Yaskawa INFORM job: miniTRJ1.JBI

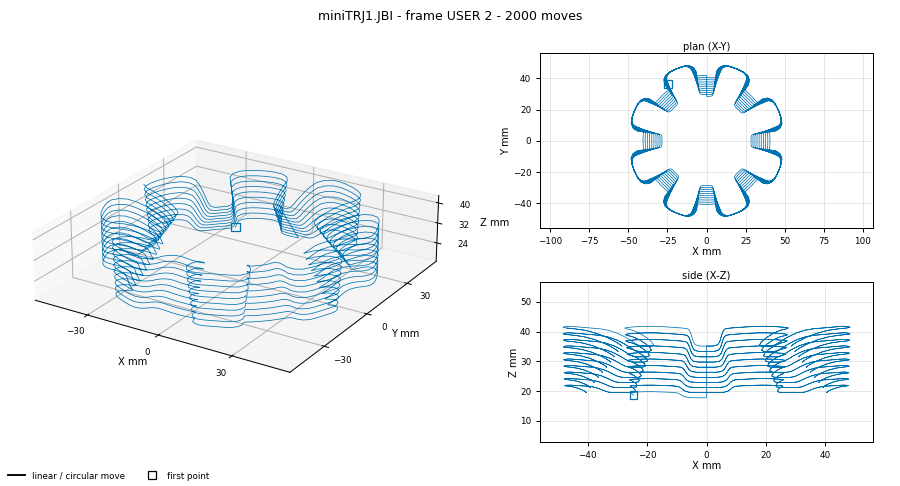
[picture p0: tool path of miniTRJ1.JBI in frame USER 2, 2000 of 2000 moves have a stored position in this frame; points joined in program order, loops and branches not executed]
/JOB
//NAME miniTRJ1
//POS
///NPOS 2000,0,0,0,0,0
///USER 2
///TOOL 1
///POSTYPE USER
///RECTAN
///RCONF 1,0,0,0,0,0,0,0,0,0,0,0,0,0,0,0,0,0,0,0,0,0,0,0
C00000=-24.565,36.346,18.587,149.9743,26.1112,0.0000
C00001=-24.917,37.674,19.017,150.2354,26.3005,0.0000
C00002=-25.352,39.110,19.349,150.5147,26.4843,0.0000
C00003=-25.558,40.564,19.514,150.8908,26.7171,0.0000
C00004=-25.030,42.161,19.602,151.6066,27.1530,0.0000
C00005=-23.802,43.680,19.673,152.6260,27.7246,0.0000
C00006=-22.056,44.839,19.746,153.7921,28.3103,0.0000
C00007=-20.124,45.768,19.794,154.9993,28.8341,0.0000
C00008=-18.133,46.592,19.794,142.7917,-4.5441,0.0000
C00009=-16.110,47.302,19.746,142.3101,-3.4636,0.0000
C00010=-14.056,47.717,19.673,141.8819,-2.3591,0.0000
C00011=-12.113,47.511,19.602,141.5332,-1.3473,0.0000
C00012=-10.611,46.755,19.514,141.3028,-0.6097,0.0000
C00013=-9.729,45.582,19.349,141.1816,-0.2190,0.0000
C00014=-9.020,44.258,19.017,141.0972,0.0798,0.0000
C00015=-8.331,43.070,18.587,141.0282,0.3730,0.0000
C00016=-7.515,42.203,18.169,140.9603,0.7327,0.0000
C00017=-6.279,41.769,17.866,140.8792,1.2870,0.0000
C00018=-4.265,41.794,17.745,140.7992,2.1565,0.0000
C00019=-2.165,41.942,17.740,140.7561,2.2344,0.0000
C00020=0.000,41.999,17.743,140.7155,0.0000,0.0000
C00021=0.000,40.651,19.482,140.7232,-0.0001,0.0000
C00022=2.042,40.599,19.478,140.7635,-2.2095,0.0000
C00023=4.057,40.463,19.484,140.8042,-2.1342,0.0000
C00024=6.024,40.479,19.630,140.8788,-1.2626,0.0000
C00025=7.200,41.019,19.996,140.9503,-0.7256,0.0000
C00026=7.966,42.055,20.504,141.0054,-0.3851,0.0000
C00027=8.617,43.471,21.031,141.0580,-0.1082,0.0000
C00028=9.290,45.059,21.441,141.1226,0.1718,0.0000
C00029=10.130,46.493,21.645,141.2220,0.5412,0.0000
C00030=11.658,47.456,21.754,141.4422,1.3035,0.0000
C00031=13.694,47.783,21.842,141.8027,2.3891,0.0000
C00032=15.881,47.377,21.932,142.2685,3.5953,0.0000
C00033=18.055,46.622,21.992,142.8073,4.7822,0.0000
C00034=20.200,45.734,21.992,155.1879,-29.0064,0.0000
C00035=22.271,44.730,21.932,153.8509,-28.4383,0.0000
C00036=24.104,43.471,21.842,152.5777,-27.7977,0.0000
C00037=25.313,41.801,21.754,151.4959,-27.1752,0.0000
C00038=25.713,40.038,21.645,150.7724,-26.7131,0.0000
C00039=25.293,38.430,21.441,150.4304,-26.4834,0.0000
C00040=24.645,36.832,21.031,150.1814,-26.3021,0.0000
C00041=24.105,35.370,20.504,149.9459,-26.1155,0.0000
C00042=23.913,34.096,19.996,149.6659,-25.8796,0.0000
C00043=24.363,32.883,19.630,149.2400,-25.4973,0.0000
C00044=25.743,31.481,19.484,148.5910,-24.8491,0.0000
C00045=27.264,30.151,19.478,148.5053,-24.8136,0.0000
C00046=28.745,28.745,19.482,149.9599,-26.5927,0.0000
C00047=30.151,27.264,19.478,151.5319,-28.3065,0.0000
C00048=31.481,25.743,19.484,151.5148,-28.2220,0.0000
C00049=32.883,24.363,19.630,150.9696,-27.4920,0.0000
C00050=34.096,23.913,19.996,150.6600,-27.0254,0.0000
C00051=35.370,24.105,20.504,150.4735,-26.7233,0.0000
C00052=36.832,24.645,21.031,150.3294,-26.4725,0.0000
C00053=38.430,25.293,21.441,150.1946,-26.2119,0.0000
C00054=40.038,25.713,21.645,150.0299,-25.8591,0.0000
C00055=41.801,25.313,21.754,149.7065,-25.1215,0.0000
C00056=43.471,24.104,21.842,149.2928,-24.0413,0.0000
C00057=44.730,22.271,21.932,148.8969,-22.8008,0.0000
C00058=45.734,20.200,21.992,148.5817,-21.5311,0.0000
C00059=46.622,18.055,21.992,-174.0048,-37.0415,0.0000
C00060=47.377,15.881,21.932,-175.4577,-37.6443,0.0000
C00061=47.783,13.694,21.842,-176.9610,-38.1581,0.0000
C00062=47.456,11.658,21.754,-178.3333,-38.5460,0.0000
C00063=46.493,10.130,21.645,-179.3058,-38.7759,0.0000
C00064=45.059,9.290,21.441,-179.7793,-38.8772,0.0000
C00065=43.471,8.617,21.031,179.8609,-38.9419,0.0000
C00066=42.055,7.966,20.504,179.5045,-38.9936,0.0000
C00067=41.019,7.200,19.996,179.0656,-39.0459,0.0000
C00068=40.479,6.024,19.630,178.3727,-39.1099,0.0000
C00069=40.463,4.057,19.484,177.2470,-39.1634,0.0000
C00070=40.599,2.042,19.478,177.1484,-39.2017,0.0000
C00071=40.651,0.000,19.482,179.9999,-39.2768,0.0000
C00072=40.599,-2.042,19.478,-177.1486,-39.2018,0.0000
C00073=40.463,-4.057,19.484,-177.2476,-39.1634,0.0000
C00074=40.479,-6.024,19.630,-178.3733,-39.1099,0.0000
C00075=41.019,-7.200,19.996,-179.0662,-39.0459,0.0000
C00076=42.055,-7.966,20.504,-179.5050,-38.9935,0.0000
C00077=43.471,-8.617,21.031,-179.8615,-38.9419,0.0000
C00078=45.059,-9.290,21.441,179.7788,-38.8771,0.0000
C00079=46.493,-10.130,21.645,179.3053,-38.7759,0.0000
C00080=47.456,-11.658,21.754,178.3329,-38.5459,0.0000
C00081=47.783,-13.694,21.842,176.9608,-38.1581,0.0000
C00082=47.377,-15.881,21.932,175.4576,-37.6442,0.0000
C00083=46.622,-18.055,21.992,174.0048,-37.0415,0.0000
C00084=45.734,-20.200,21.992,-148.5817,-21.5311,0.0000
C00085=44.730,-22.271,21.932,-148.8969,-22.8008,0.0000
C00086=43.471,-24.104,21.842,-149.2929,-24.0415,0.0000
C00087=41.801,-25.313,21.754,-149.7066,-25.1217,0.0000
C00088=40.038,-25.713,21.645,-150.0301,-25.8595,0.0000
C00089=38.430,-25.293,21.441,-150.1948,-26.2122,0.0000
C00090=36.832,-24.645,21.031,-150.3297,-26.4729,0.0000
C00091=35.370,-24.105,20.504,-150.4737,-26.7237,0.0000
C00092=34.096,-23.913,19.996,-150.6602,-27.0258,0.0000
C00093=32.883,-24.363,19.630,-150.9699,-27.4924,0.0000
C00094=31.481,-25.743,19.484,-151.5151,-28.2224,0.0000
C00095=30.151,-27.264,19.478,-151.5321,-28.3066,0.0000
C00096=28.745,-28.745,19.482,-149.9600,-26.5929,0.0000
C00097=27.264,-30.151,19.478,-148.5053,-24.8138,0.0000
C00098=25.743,-31.481,19.484,-148.5913,-24.8495,0.0000
C00099=24.363,-32.883,19.630,-149.2404,-25.4977,0.0000
C00100=23.913,-34.096,19.996,-149.6663,-25.8800,0.0000
C00101=24.105,-35.370,20.504,-149.9463,-26.1158,0.0000
C00102=24.645,-36.832,21.031,-150.1818,-26.3024,0.0000
C00103=25.293,-38.430,21.441,-150.4307,-26.4836,0.0000
C00104=25.713,-40.038,21.645,-150.7727,-26.7133,0.0000
C00105=25.313,-41.801,21.754,-151.4962,-27.1754,0.0000
C00106=24.104,-43.471,21.842,-152.5779,-27.7978,0.0000
C00107=22.271,-44.730,21.932,-153.8509,-28.4383,0.0000
C00108=20.200,-45.734,21.992,-155.1879,-29.0063,0.0000
C00109=18.055,-46.622,21.992,-142.8073,4.7822,0.0000
C00110=15.881,-47.377,21.932,-142.2685,3.5953,0.0000
C00111=13.694,-47.783,21.842,-141.8027,2.3891,0.0000
C00112=11.658,-47.456,21.754,-141.4422,1.3035,0.0000
C00113=10.130,-46.493,21.645,-141.2220,0.5412,0.0000
C00114=9.290,-45.059,21.441,-141.1226,0.1718,0.0000
C00115=8.617,-43.471,21.031,-141.0580,-0.1082,0.0000
C00116=7.966,-42.055,20.504,-141.0054,-0.3851,0.0000
C00117=7.200,-41.019,19.996,-140.9503,-0.7256,0.0000
C00118=6.024,-40.479,19.630,-140.8788,-1.2626,0.0000
C00119=4.057,-40.463,19.484,-140.8042,-2.1342,0.0000
C00120=2.042,-40.599,19.478,-140.7635,-2.2095,0.0000
C00121=0.000,-40.651,19.482,-140.7232,-0.0001,0.0000
C00122=0.000,-40.651,19.482,-140.7232,-0.0001,0.0000
C00123=-2.042,-40.599,19.478,-140.7635,2.2093,0.0000
C00124=-4.057,-40.463,19.484,-140.8042,2.1337,0.0000
C00125=-6.024,-40.479,19.630,-140.8788,1.2621,0.0000
C00126=-7.200,-41.019,19.996,-140.9504,0.7252,0.0000
C00127=-7.966,-42.055,20.504,-141.0054,0.3847,0.0000
C00128=-8.617,-43.471,21.031,-141.0581,0.1077,0.0000
C00129=-9.290,-45.059,21.441,-141.1227,-0.1722,0.0000
C00130=-10.130,-46.493,21.645,-141.2221,-0.5416,0.0000
C00131=-11.658,-47.456,21.754,-141.4423,-1.3038,0.0000
C00132=-13.694,-47.783,21.842,-141.8027,-2.3893,0.0000
C00133=-15.881,-47.377,21.932,-142.2685,-3.5953,0.0000
C00134=-18.055,-46.622,21.992,-142.8073,-4.7822,0.0000
C00135=-20.200,-45.734,21.992,-155.1879,29.0064,0.0000
C00136=-22.271,-44.730,21.932,-153.8509,28.4383,0.0000
C00137=-24.104,-43.471,21.842,-152.5777,27.7977,0.0000
C00138=-25.313,-41.801,21.754,-151.4959,27.1752,0.0000
C00139=-25.713,-40.038,21.645,-150.7724,26.7131,0.0000
C00140=-25.293,-38.430,21.441,-150.4304,26.4834,0.0000
C00141=-24.645,-36.832,21.031,-150.1814,26.3021,0.0000
C00142=-24.105,-35.370,20.504,-149.9459,26.1155,0.0000
C00143=-23.913,-34.096,19.996,-149.6659,25.8796,0.0000
C00144=-24.363,-32.883,19.630,-149.2400,25.4973,0.0000
C00145=-25.743,-31.481,19.484,-148.5910,24.8491,0.0000
C00146=-27.264,-30.151,19.478,-148.5053,24.8136,0.0000
C00147=-28.745,-28.745,19.482,-149.9599,26.5927,0.0000
C00148=-30.151,-27.264,19.478,-151.5319,28.3065,0.0000
C00149=-31.481,-25.743,19.484,-151.5148,28.2220,0.0000
C00150=-32.883,-24.363,19.630,-150.9696,27.4920,0.0000
C00151=-34.096,-23.913,19.996,-150.6600,27.0254,0.0000
C00152=-35.370,-24.105,20.504,-150.4735,26.7233,0.0000
C00153=-36.832,-24.645,21.031,-150.3294,26.4725,0.0000
C00154=-38.430,-25.293,21.441,-150.1946,26.2119,0.0000
C00155=-40.038,-25.713,21.645,-150.0299,25.8591,0.0000
C00156=-41.801,-25.313,21.754,-149.7065,25.1215,0.0000
C00157=-43.471,-24.104,21.842,-149.2928,24.0413,0.0000
C00158=-44.730,-22.271,21.932,-148.8969,22.8008,0.0000
C00159=-45.734,-20.200,21.992,-148.5817,21.5311,0.0000
C00160=-46.622,-18.055,21.992,174.0048,37.0415,0.0000
C00161=-47.377,-15.881,21.932,175.4577,37.6443,0.0000
C00162=-47.783,-13.694,21.842,176.9610,38.1581,0.0000
C00163=-47.456,-11.658,21.754,178.3333,38.5460,0.0000
C00164=-46.493,-10.130,21.645,179.3058,38.7759,0.0000
C00165=-45.059,-9.290,21.441,179.7793,38.8772,0.0000
C00166=-43.471,-8.617,21.031,-179.8609,38.9419,0.0000
C00167=-42.055,-7.966,20.504,-179.5045,38.9936,0.0000
C00168=-41.019,-7.200,19.996,-179.0656,39.0459,0.0000
C00169=-40.479,-6.024,19.630,-178.3727,39.1099,0.0000
C00170=-40.463,-4.057,19.484,-177.2470,39.1634,0.0000
C00171=-40.599,-2.042,19.478,-177.1484,39.2017,0.0000
C00172=-40.651,0.000,19.482,-179.9999,39.2768,0.0000
C00173=-40.599,2.042,19.478,177.1486,39.2018,0.0000
C00174=-40.463,4.057,19.484,177.2476,39.1634,0.0000
C00175=-40.479,6.024,19.630,178.3733,39.1099,0.0000
C00176=-41.019,7.200,19.996,179.0662,39.0459,0.0000
C00177=-42.055,7.966,20.504,179.5050,38.9935,0.0000
C00178=-43.471,8.617,21.031,179.8615,38.9419,0.0000
C00179=-45.059,9.290,21.441,-179.7788,38.8771,0.0000
C00180=-46.493,10.130,21.645,-179.3053,38.7759,0.0000
C00181=-47.456,11.658,21.754,-178.3329,38.5459,0.0000
C00182=-47.783,13.694,21.842,-176.9608,38.1581,0.0000
C00183=-47.377,15.881,21.932,-175.4576,37.6442,0.0000
C00184=-46.622,18.055,21.992,-174.0048,37.0415,0.0000
C00185=-45.734,20.200,21.992,148.5817,21.5311,0.0000
C00186=-44.730,22.271,21.932,148.8969,22.8008,0.0000
C00187=-43.471,24.104,21.842,149.2929,24.0415,0.0000
C00188=-41.801,25.313,21.754,149.7066,25.1217,0.0000
C00189=-40.038,25.713,21.645,150.0301,25.8595,0.0000
C00190=-38.430,25.293,21.441,150.1948,26.2122,0.0000
C00191=-36.832,24.645,21.031,150.3297,26.4729,0.0000
C00192=-35.370,24.105,20.504,150.4737,26.7237,0.0000
C00193=-34.096,23.913,19.996,150.6602,27.0258,0.0000
C00194=-32.883,24.363,19.630,150.9699,27.4924,0.0000
C00195=-31.481,25.743,19.484,151.5151,28.2224,0.0000
C00196=-30.151,27.264,19.478,151.5321,28.3066,0.0000
C00197=-28.745,28.745,19.482,149.9600,26.5929,0.0000
C00198=-27.264,30.151,19.478,148.5053,24.8138,0.0000
C00199=-25.743,31.481,19.484,148.5913,24.8495,0.0000
C00200=-24.363,32.883,19.630,149.2404,25.4977,0.0000
C00201=-23.913,34.096,19.996,149.6663,25.8800,0.0000
C00202=-24.105,35.370,20.504,149.9463,26.1158,0.0000
C00203=-24.645,36.832,21.031,150.1818,26.3024,0.0000
C00204=-25.293,38.430,21.441,150.4307,26.4836,0.0000
C00205=-25.713,40.038,21.645,150.7727,26.7133,0.0000
C00206=-25.313,41.801,21.754,151.4962,27.1754,0.0000
C00207=-24.104,43.471,21.842,152.5779,27.7978,0.0000
C00208=-22.271,44.730,21.932,153.8509,28.4383,0.0000
C00209=-20.200,45.734,21.992,155.1879,29.0063,0.0000
C00210=-18.055,46.622,21.992,142.8073,-4.7822,0.0000
C00211=-15.881,47.377,21.932,142.2685,-3.5953,0.0000
C00212=-13.694,47.783,21.842,141.8027,-2.3893,0.0000
C00213=-11.658,47.456,21.754,141.4423,-1.3038,0.0000
C00214=-10.130,46.493,21.645,141.2221,-0.5416,0.0000
C00215=-9.290,45.059,21.441,141.1227,-0.1722,0.0000
C00216=-8.617,43.471,21.031,141.0581,0.1077,0.0000
C00217=-7.966,42.055,20.504,141.0054,0.3847,0.0000
C00218=-7.200,41.019,19.996,140.9504,0.7252,0.0000
C00219=-6.024,40.479,19.630,140.8788,1.2621,0.0000
C00220=-4.057,40.463,19.484,140.8042,2.1337,0.0000
C00221=-2.042,40.599,19.478,140.7635,2.2093,0.0000
C00222=0.000,40.651,19.482,140.7232,-0.0001,0.0000
C00223=0.000,39.279,21.202,140.7756,-0.0003,0.0000
C00224=1.916,39.231,21.197,140.8155,-2.1795,0.0000
C00225=3.846,39.107,21.204,140.8539,-2.1148,0.0000
C00226=5.765,39.166,21.375,140.9231,-1.2456,0.0000
C00227=6.881,39.812,21.808,140.9851,-0.7291,0.0000
C00228=7.594,41.021,22.410,141.0266,-0.4101,0.0000
C00229=8.207,42.669,23.038,141.0611,-0.1507,0.0000
C00230=8.843,44.528,23.528,141.1028,0.1103,0.0000
C00231=9.641,46.227,23.773,141.1765,0.4563,0.0000
C00232=11.196,47.401,23.904,141.3824,1.2437,0.0000
C00233=13.327,47.850,24.010,141.7525,2.4066,0.0000
C00234=15.648,47.454,24.119,142.2575,3.7194,0.0000
C00235=17.976,46.653,24.190,142.8578,5.0171,0.0000
C00236=20.278,45.699,24.190,155.4053,-29.1535,0.0000
C00237=22.491,44.620,24.119,153.9310,-28.5410,0.0000
C00238=24.412,43.258,24.010,152.5460,-27.8428,0.0000
C00239=25.601,41.434,23.904,151.4015,-27.1655,0.0000
C00240=25.871,39.504,23.773,150.6737,-26.6744,0.0000
C00241=25.233,37.739,23.528,150.3706,-26.4471,0.0000
C00242=24.369,35.974,23.038,150.1550,-26.2666,0.0000
C00243=23.637,34.376,22.410,149.9476,-26.0828,0.0000
C00244=23.286,33.017,21.808,149.6942,-25.8557,0.0000
C00245=23.618,31.771,21.375,149.2905,-25.4839,0.0000
C00246=24.933,30.373,21.204,148.6476,-24.8345,0.0000
C00247=26.385,29.096,21.197,148.5708,-24.8062,0.0000
C00248=27.774,27.774,21.202,150.0061,-26.5605,0.0000
C00249=29.096,26.385,21.197,151.5569,-28.2507,0.0000
C00250=30.373,24.933,21.204,151.5453,-28.1759,0.0000
C00251=31.771,23.618,21.375,150.9969,-27.4512,0.0000
C00252=33.017,23.286,21.808,150.6931,-27.0067,0.0000
C00253=34.376,23.637,22.410,150.5094,-26.7299,0.0000
C00254=35.974,24.369,23.038,150.3614,-26.5042,0.0000
C00255=37.739,25.233,23.528,150.2192,-26.2726,0.0000
C00256=39.504,25.871,23.773,150.0477,-25.9541,0.0000
C00257=41.434,25.601,23.904,149.6945,-25.2054,0.0000
C00258=43.258,24.412,24.010,149.2375,-24.0580,0.0000
C00259=44.620,22.491,24.119,148.8059,-22.7088,0.0000
C00260=45.699,20.278,24.190,148.4720,-21.3136,0.0000
C00261=46.653,17.976,24.190,-173.7153,-36.9761,0.0000
C00262=47.454,15.648,24.119,-175.3005,-37.6491,0.0000
C00263=47.850,13.327,24.010,-176.9367,-38.2077,0.0000
C00264=47.401,11.196,23.904,-178.4084,-38.6068,0.0000
C00265=46.227,9.641,23.773,-179.4143,-38.8221,0.0000
C00266=44.528,8.843,23.528,-179.8583,-38.8971,0.0000
C00267=42.669,8.207,23.038,179.8062,-38.9387,0.0000
C00268=41.021,7.594,22.410,179.4725,-38.9722,0.0000
C00269=39.812,6.881,21.808,179.0616,-39.0111,0.0000
C00270=39.166,5.765,21.375,178.3957,-39.0659,0.0000
C00271=39.107,3.846,21.204,177.2739,-39.1143,0.0000
C00272=39.231,1.916,21.197,177.1891,-39.1508,0.0000
C00273=39.279,0.000,21.202,179.9997,-39.2244,0.0000
C00274=39.231,-1.916,21.197,-177.1893,-39.1508,0.0000
C00275=39.107,-3.847,21.204,-177.2745,-39.1143,0.0000
C00276=39.166,-5.765,21.375,-178.3963,-39.0659,0.0000
C00277=39.812,-6.881,21.808,-179.0622,-39.0111,0.0000
C00278=41.021,-7.594,22.410,-179.4731,-38.9722,0.0000
C00279=42.669,-8.207,23.038,-179.8067,-38.9387,0.0000
C00280=44.528,-8.843,23.528,179.8578,-38.8971,0.0000
C00281=46.227,-9.641,23.773,179.4138,-38.8220,0.0000
C00282=47.401,-11.196,23.904,178.4081,-38.6067,0.0000
C00283=47.850,-13.327,24.010,176.9365,-38.2077,0.0000
C00284=47.454,-15.648,24.119,175.3004,-37.6491,0.0000
C00285=46.653,-17.976,24.190,173.7153,-36.9761,0.0000
C00286=45.699,-20.278,24.190,-148.4719,-21.3136,0.0000
C00287=44.620,-22.491,24.119,-148.8059,-22.7088,0.0000
C00288=43.258,-24.412,24.010,-149.2376,-24.0581,0.0000
C00289=41.434,-25.601,23.904,-149.6946,-25.2056,0.0000
C00290=39.504,-25.871,23.773,-150.0479,-25.9544,0.0000
C00291=37.739,-25.233,23.528,-150.2194,-26.2730,0.0000
C00292=35.974,-24.369,23.038,-150.3617,-26.5046,0.0000
C00293=34.376,-23.637,22.410,-150.5096,-26.7303,0.0000
C00294=33.017,-23.286,21.808,-150.6934,-27.0071,0.0000
C00295=31.771,-23.618,21.375,-150.9972,-27.4516,0.0000
C00296=30.373,-24.933,21.204,-151.5456,-28.1763,0.0000
C00297=29.096,-26.385,21.197,-151.5571,-28.2508,0.0000
C00298=27.774,-27.774,21.202,-150.0065,-26.5609,0.0000
C00299=26.385,-29.096,21.197,-148.5708,-24.8064,0.0000
C00300=24.933,-30.373,21.204,-148.6479,-24.8349,0.0000
C00301=23.618,-31.771,21.375,-149.2908,-25.4843,0.0000
C00302=23.286,-33.017,21.808,-149.6945,-25.8560,0.0000
C00303=23.637,-34.376,22.410,-149.9479,-26.0831,0.0000
C00304=24.369,-35.974,23.038,-150.1554,-26.2669,0.0000
C00305=25.233,-37.739,23.528,-150.3710,-26.4473,0.0000
C00306=25.871,-39.504,23.773,-150.6740,-26.6747,0.0000
C00307=25.601,-41.434,23.904,-151.4017,-27.1657,0.0000
C00308=24.412,-43.258,24.010,-152.5461,-27.8429,0.0000
C00309=22.491,-44.620,24.119,-153.9311,-28.5411,0.0000
C00310=20.278,-45.699,24.190,-155.4053,-29.1535,0.0000
C00311=17.976,-46.653,24.190,-142.8578,5.0171,0.0000
C00312=15.648,-47.454,24.119,-142.2575,3.7194,0.0000
C00313=13.327,-47.850,24.010,-141.7525,2.4066,0.0000
C00314=11.196,-47.401,23.904,-141.3824,1.2437,0.0000
C00315=9.641,-46.227,23.773,-141.1765,0.4563,0.0000
C00316=8.843,-44.528,23.528,-141.1028,0.1103,0.0000
C00317=8.207,-42.669,23.038,-141.0611,-0.1507,0.0000
C00318=7.594,-41.021,22.410,-141.0266,-0.4101,0.0000
C00319=6.881,-39.812,21.808,-140.9851,-0.7291,0.0000
C00320=5.765,-39.166,21.375,-140.9231,-1.2456,0.0000
C00321=3.846,-39.107,21.204,-140.8539,-2.1148,0.0000
C00322=1.916,-39.231,21.197,-140.8155,-2.1795,0.0000
C00323=0.000,-39.279,21.202,-140.7756,-0.0003,0.0000
C00324=0.000,-39.279,21.202,-140.7756,-0.0003,0.0000
C00325=-1.916,-39.231,21.197,-140.8154,2.1793,0.0000
C00326=-3.847,-39.107,21.204,-140.8539,2.1143,0.0000
C00327=-5.765,-39.166,21.375,-140.9231,1.2451,0.0000
C00328=-6.881,-39.812,21.808,-140.9852,0.7287,0.0000
C00329=-7.594,-41.021,22.410,-141.0266,0.4096,0.0000
C00330=-8.207,-42.669,23.038,-141.0611,0.1503,0.0000
C00331=-8.843,-44.528,23.528,-141.1028,-0.1107,0.0000
C00332=-9.641,-46.227,23.773,-141.1765,-0.4567,0.0000
C00333=-11.196,-47.401,23.904,-141.3825,-1.2439,0.0000
C00334=-13.327,-47.850,24.010,-141.7525,-2.4068,0.0000
C00335=-15.648,-47.454,24.119,-142.2575,-3.7194,0.0000
C00336=-17.976,-46.653,24.190,-142.8578,-5.0171,0.0000
C00337=-20.278,-45.699,24.190,-155.4053,29.1535,0.0000
C00338=-22.491,-44.620,24.119,-153.9310,28.5410,0.0000
C00339=-24.412,-43.258,24.010,-152.5460,27.8428,0.0000
C00340=-25.601,-41.434,23.904,-151.4015,27.1655,0.0000
C00341=-25.871,-39.504,23.773,-150.6737,26.6744,0.0000
C00342=-25.233,-37.739,23.528,-150.3706,26.4471,0.0000
C00343=-24.369,-35.974,23.038,-150.1550,26.2666,0.0000
C00344=-23.637,-34.376,22.410,-149.9476,26.0828,0.0000
C00345=-23.286,-33.017,21.808,-149.6942,25.8557,0.0000
C00346=-23.618,-31.771,21.375,-149.2905,25.4839,0.0000
C00347=-24.933,-30.373,21.204,-148.6476,24.8345,0.0000
C00348=-26.385,-29.096,21.197,-148.5708,24.8062,0.0000
C00349=-27.774,-27.774,21.202,-150.0061,26.5605,0.0000
C00350=-29.096,-26.385,21.197,-151.5569,28.2507,0.0000
C00351=-30.373,-24.933,21.204,-151.5453,28.1759,0.0000
C00352=-31.771,-23.618,21.375,-150.9969,27.4512,0.0000
C00353=-33.017,-23.286,21.808,-150.6931,27.0067,0.0000
C00354=-34.376,-23.637,22.410,-150.5094,26.7299,0.0000
C00355=-35.974,-24.369,23.038,-150.3614,26.5042,0.0000
C00356=-37.739,-25.233,23.528,-150.2192,26.2726,0.0000
C00357=-39.504,-25.871,23.773,-150.0477,25.9541,0.0000
C00358=-41.434,-25.601,23.904,-149.6945,25.2054,0.0000
C00359=-43.258,-24.412,24.010,-149.2375,24.0580,0.0000
C00360=-44.620,-22.491,24.119,-148.8059,22.7088,0.0000
C00361=-45.699,-20.278,24.190,-148.4720,21.3136,0.0000
C00362=-46.653,-17.976,24.190,173.7153,36.9761,0.0000
C00363=-47.454,-15.648,24.119,175.3005,37.6491,0.0000
C00364=-47.850,-13.327,24.010,176.9367,38.2077,0.0000
C00365=-47.401,-11.196,23.904,178.4084,38.6068,0.0000
C00366=-46.227,-9.641,23.773,179.4143,38.8221,0.0000
C00367=-44.528,-8.843,23.528,179.8583,38.8971,0.0000
C00368=-42.669,-8.207,23.038,-179.8062,38.9387,0.0000
C00369=-41.021,-7.594,22.410,-179.4725,38.9722,0.0000
C00370=-39.812,-6.881,21.808,-179.0616,39.0111,0.0000
C00371=-39.166,-5.765,21.375,-178.3957,39.0659,0.0000
C00372=-39.107,-3.846,21.204,-177.2739,39.1143,0.0000
C00373=-39.231,-1.916,21.197,-177.1891,39.1508,0.0000
C00374=-39.279,0.000,21.202,-179.9997,39.2244,0.0000
C00375=-39.231,1.916,21.197,177.1893,39.1508,0.0000
C00376=-39.107,3.847,21.204,177.2745,39.1143,0.0000
C00377=-39.166,5.765,21.375,178.3963,39.0659,0.0000
C00378=-39.812,6.881,21.808,179.0622,39.0111,0.0000
C00379=-41.021,7.594,22.410,179.4731,38.9722,0.0000
C00380=-42.669,8.207,23.038,179.8067,38.9387,0.0000
C00381=-44.528,8.843,23.528,-179.8578,38.8971,0.0000
C00382=-46.227,9.641,23.773,-179.4138,38.8220,0.0000
C00383=-47.401,11.196,23.904,-178.4081,38.6067,0.0000
C00384=-47.850,13.327,24.010,-176.9365,38.2077,0.0000
C00385=-47.454,15.648,24.119,-175.3004,37.6491,0.0000
C00386=-46.653,17.976,24.190,-173.7153,36.9761,0.0000
C00387=-45.699,20.278,24.190,148.4719,21.3136,0.0000
C00388=-44.620,22.491,24.119,148.8059,22.7088,0.0000
C00389=-43.258,24.412,24.010,149.2376,24.0581,0.0000
C00390=-41.434,25.601,23.904,149.6946,25.2056,0.0000
C00391=-39.504,25.871,23.773,150.0479,25.9544,0.0000
C00392=-37.739,25.233,23.528,150.2194,26.2730,0.0000
C00393=-35.974,24.369,23.038,150.3617,26.5046,0.0000
C00394=-34.376,23.637,22.410,150.5096,26.7303,0.0000
C00395=-33.017,23.286,21.808,150.6934,27.0071,0.0000
C00396=-31.771,23.618,21.375,150.9972,27.4516,0.0000
C00397=-30.373,24.933,21.204,151.5456,28.1763,0.0000
C00398=-29.096,26.385,21.197,151.5571,28.2508,0.0000
C00399=-27.774,27.774,21.202,150.0065,26.5609,0.0000
C00400=-26.385,29.096,21.197,148.5708,24.8064,0.0000
C00401=-24.933,30.373,21.204,148.6479,24.8349,0.0000
C00402=-23.618,31.771,21.375,149.2908,25.4843,0.0000
C00403=-23.286,33.017,21.808,149.6945,25.8560,0.0000
C00404=-23.637,34.376,22.410,149.9479,26.0831,0.0000
C00405=-24.369,35.974,23.038,150.1554,26.2669,0.0000
C00406=-25.233,37.739,23.528,150.3710,26.4473,0.0000
C00407=-25.871,39.504,23.773,150.6740,26.6747,0.0000
C00408=-25.601,41.434,23.904,151.4017,27.1657,0.0000
C00409=-24.412,43.258,24.010,152.5461,27.8429,0.0000
C00410=-22.491,44.620,24.119,153.9311,28.5411,0.0000
C00411=-20.278,45.699,24.190,155.4053,29.1535,0.0000
C00412=-17.976,46.653,24.190,142.8578,-5.0171,0.0000
C00413=-15.648,47.454,24.119,142.2575,-3.7194,0.0000
C00414=-13.327,47.850,24.010,141.7525,-2.4068,0.0000
C00415=-11.196,47.401,23.904,141.3825,-1.2439,0.0000
C00416=-9.641,46.227,23.773,141.1765,-0.4567,0.0000
C00417=-8.843,44.528,23.528,141.1028,-0.1107,0.0000
C00418=-8.207,42.669,23.038,141.0611,0.1503,0.0000
C00419=-7.594,41.021,22.410,141.0266,0.4096,0.0000
C00420=-6.881,39.812,21.808,140.9852,0.7287,0.0000
C00421=-5.765,39.166,21.375,140.9231,1.2451,0.0000
C00422=-3.847,39.107,21.204,140.8539,2.1143,0.0000
C00423=-1.916,39.231,21.197,140.8154,2.1793,0.0000
C00424=0.000,39.279,21.202,140.7756,-0.0003,0.0000
C00425=0.000,37.892,22.909,140.8700,-0.0004,0.0000
C00426=1.790,37.849,22.904,140.9092,-2.1449,0.0000
C00427=3.633,37.737,22.912,140.9457,-2.0985,0.0000
C00428=5.504,37.838,23.110,141.0095,-1.2353,0.0000
C00429=6.557,38.594,23.612,141.0620,-0.7420,0.0000
C00430=7.219,39.979,24.311,141.0895,-0.4460,0.0000
C00431=7.794,41.862,25.043,141.1044,-0.2054,0.0000
C00432=8.395,43.994,25.615,141.1205,0.0368,0.0000
C00433=9.151,45.960,25.902,141.1649,0.3590,0.0000
C00434=10.734,47.345,26.054,141.3528,1.1718,0.0000
C00435=12.959,47.917,26.178,141.7303,2.4150,0.0000
C00436=15.415,47.531,26.305,142.2760,3.8384,0.0000
C00437=17.897,46.683,26.389,142.9419,5.2501,0.0000
C00438=20.355,45.665,26.389,155.6510,-29.2771,0.0000
C00439=22.710,44.510,26.305,154.0336,-28.6211,0.0000
C00440=24.719,43.046,26.178,152.5325,-27.8632,0.0000
C00441=25.888,41.068,26.054,151.3253,-27.1275,0.0000
C00442=26.028,38.969,25.902,150.5964,-26.6049,0.0000
C00443=25.172,37.045,25.615,150.3357,-26.3782,0.0000
C00444=24.090,35.112,25.043,150.1558,-26.1969,0.0000
C00445=23.165,33.374,24.311,149.9784,-26.0158,0.0000
C00446=22.654,31.927,23.612,149.7531,-25.7985,0.0000
C00447=22.864,30.647,23.110,149.3733,-25.4395,0.0000
C00448=24.115,29.253,22.912,148.7389,-24.7921,0.0000
C00449=25.498,28.029,22.904,148.6760,-24.7771,0.0000
C00450=26.793,26.793,22.909,150.0894,-26.5025,0.0000
C00451=28.029,25.498,22.904,151.6157,-28.1654,0.0000
C00452=29.253,24.115,22.912,151.6151,-28.1060,0.0000
C00453=30.647,22.864,23.110,151.0663,-27.3897,0.0000
C00454=31.927,22.654,23.612,150.7699,-26.9694,0.0000
C00455=33.374,23.165,24.311,150.5897,-26.7195,0.0000
C00456=35.112,24.090,25.043,150.4371,-26.5206,0.0000
C00457=37.045,25.172,25.615,150.2851,-26.3198,0.0000
C00458=38.969,26.028,25.902,150.1039,-26.0381,0.0000
C00459=41.068,25.888,26.054,149.7171,-25.2803,0.0000
C00460=43.046,24.719,26.178,149.2127,-24.0648,0.0000
C00461=44.510,22.710,26.305,148.7436,-22.6029,0.0000
C00462=45.665,20.355,26.389,148.3924,-21.0774,0.0000
C00463=46.683,17.897,26.389,-173.4316,-36.8768,0.0000
C00464=47.531,15.415,26.305,-175.1515,-37.6247,0.0000
C00465=47.917,12.959,26.178,-176.9251,-38.2295,0.0000
C00466=47.345,10.734,26.054,-178.4998,-38.6376,0.0000
C00467=45.960,9.151,25.902,-179.5392,-38.8342,0.0000
C00468=43.994,8.395,25.615,-179.9528,-38.8795,0.0000
C00469=41.862,7.794,25.043,179.7361,-38.8953,0.0000
C00470=39.979,7.219,24.311,179.4268,-38.9091,0.0000
C00471=38.594,6.557,23.612,179.0461,-38.9341,0.0000
C00472=37.838,5.504,23.110,178.4108,-38.9797,0.0000
C00473=37.737,3.633,22.912,177.2985,-39.0231,0.0000
C00474=37.849,1.790,22.904,177.2373,-39.0582,0.0000
C00475=37.892,0.000,22.909,179.9995,-39.1300,0.0000
C00476=37.849,-1.790,22.904,-177.2375,-39.0582,0.0000
C00477=37.737,-3.633,22.912,-177.2991,-39.0231,0.0000
C00478=37.838,-5.504,23.110,-178.4114,-38.9797,0.0000
C00479=38.594,-6.557,23.612,-179.0467,-38.9341,0.0000
C00480=39.979,-7.219,24.311,-179.4273,-38.9091,0.0000
C00481=41.862,-7.794,25.043,-179.7367,-38.8952,0.0000
C00482=43.994,-8.395,25.615,179.9523,-38.8795,0.0000
C00483=45.960,-9.151,25.902,179.5386,-38.8341,0.0000
C00484=47.345,-10.734,26.054,178.4994,-38.6375,0.0000
C00485=47.917,-12.959,26.178,176.9249,-38.2295,0.0000
C00486=47.531,-15.415,26.305,175.1514,-37.6246,0.0000
C00487=46.683,-17.897,26.389,173.4316,-36.8768,0.0000
C00488=45.665,-20.355,26.389,-148.3924,-21.0774,0.0000
C00489=44.510,-22.710,26.305,-148.7436,-22.6029,0.0000
C00490=43.046,-24.719,26.178,-149.2128,-24.0649,0.0000
C00491=41.068,-25.888,26.054,-149.7173,-25.2806,0.0000
C00492=38.969,-26.028,25.902,-150.1041,-26.0384,0.0000
C00493=37.045,-25.172,25.615,-150.2853,-26.3202,0.0000
C00494=35.112,-24.090,25.043,-150.4374,-26.5210,0.0000
C00495=33.374,-23.165,24.311,-150.5899,-26.7199,0.0000
C00496=31.927,-22.654,23.612,-150.7702,-26.9698,0.0000
C00497=30.647,-22.864,23.110,-151.0666,-27.3901,0.0000
C00498=29.253,-24.115,22.912,-151.6154,-28.1064,0.0000
C00499=28.029,-25.498,22.904,-151.6159,-28.1655,0.0000
C00500=26.793,-26.793,22.909,-150.0900,-26.5032,0.0000
C00501=25.498,-28.029,22.904,-148.6761,-24.7773,0.0000
C00502=24.115,-29.253,22.912,-148.7393,-24.7925,0.0000
C00503=22.864,-30.647,23.110,-149.3737,-25.4398,0.0000
C00504=22.654,-31.927,23.612,-149.7534,-25.7988,0.0000
C00505=23.165,-33.374,24.311,-149.9788,-26.0162,0.0000
C00506=24.090,-35.112,25.043,-150.1562,-26.1972,0.0000
C00507=25.172,-37.045,25.615,-150.3361,-26.3785,0.0000
C00508=26.028,-38.969,25.902,-150.5967,-26.6051,0.0000
C00509=25.888,-41.068,26.054,-151.3255,-27.1277,0.0000
C00510=24.719,-43.046,26.178,-152.5326,-27.8634,0.0000
C00511=22.710,-44.510,26.305,-154.0336,-28.6211,0.0000
C00512=20.355,-45.665,26.389,-155.6510,-29.2771,0.0000
C00513=17.897,-46.683,26.389,-142.9419,5.2501,0.0000
C00514=15.415,-47.531,26.305,-142.2760,3.8384,0.0000
C00515=12.959,-47.917,26.178,-141.7303,2.4150,0.0000
C00516=10.734,-47.345,26.054,-141.3528,1.1718,0.0000
C00517=9.151,-45.960,25.902,-141.1649,0.3590,0.0000
C00518=8.395,-43.994,25.615,-141.1205,0.0368,0.0000
C00519=7.794,-41.862,25.043,-141.1044,-0.2054,0.0000
C00520=7.219,-39.979,24.311,-141.0895,-0.4460,0.0000
C00521=6.557,-38.594,23.612,-141.0620,-0.7420,0.0000
C00522=5.504,-37.838,23.110,-141.0095,-1.2353,0.0000
C00523=3.633,-37.737,22.912,-140.9457,-2.0985,0.0000
C00524=1.790,-37.849,22.904,-140.9092,-2.1449,0.0000
C00525=0.000,-37.892,22.909,-140.8700,-0.0004,0.0000
C00526=0.000,-37.892,22.909,-140.8700,-0.0004,0.0000
C00527=-1.790,-37.849,22.904,-140.9092,2.1447,0.0000
C00528=-3.633,-37.737,22.912,-140.9457,2.0980,0.0000
C00529=-5.504,-37.838,23.110,-141.0096,1.2348,0.0000
C00530=-6.557,-38.594,23.612,-141.0621,0.7415,0.0000
C00531=-7.219,-39.979,24.311,-141.0895,0.4456,0.0000
C00532=-7.794,-41.862,25.043,-141.1045,0.2049,0.0000
C00533=-8.395,-43.994,25.615,-141.1205,-0.0372,0.0000
C00534=-9.151,-45.960,25.902,-141.1650,-0.3594,0.0000
C00535=-10.734,-47.345,26.054,-141.3529,-1.1721,0.0000
C00536=-12.959,-47.917,26.178,-141.7304,-2.4152,0.0000
C00537=-15.415,-47.531,26.305,-142.2760,-3.8385,0.0000
C00538=-17.897,-46.683,26.389,-142.9419,-5.2501,0.0000
C00539=-20.355,-45.665,26.389,-155.6510,29.2771,0.0000
C00540=-22.710,-44.510,26.305,-154.0336,28.6211,0.0000
C00541=-24.719,-43.046,26.178,-152.5325,27.8632,0.0000
C00542=-25.888,-41.068,26.054,-151.3253,27.1275,0.0000
C00543=-26.028,-38.969,25.902,-150.5964,26.6049,0.0000
C00544=-25.172,-37.045,25.615,-150.3357,26.3782,0.0000
C00545=-24.090,-35.112,25.043,-150.1558,26.1969,0.0000
C00546=-23.165,-33.374,24.311,-149.9784,26.0158,0.0000
C00547=-22.654,-31.927,23.612,-149.7531,25.7985,0.0000
C00548=-22.864,-30.647,23.110,-149.3733,25.4395,0.0000
C00549=-24.115,-29.253,22.912,-148.7389,24.7921,0.0000
C00550=-25.498,-28.029,22.904,-148.6760,24.7771,0.0000
C00551=-26.793,-26.793,22.909,-150.0894,26.5025,0.0000
C00552=-28.029,-25.498,22.904,-151.6157,28.1654,0.0000
C00553=-29.253,-24.115,22.912,-151.6151,28.1060,0.0000
C00554=-30.647,-22.864,23.110,-151.0663,27.3897,0.0000
C00555=-31.927,-22.654,23.612,-150.7699,26.9694,0.0000
C00556=-33.374,-23.165,24.311,-150.5897,26.7195,0.0000
C00557=-35.112,-24.090,25.043,-150.4371,26.5206,0.0000
C00558=-37.045,-25.172,25.615,-150.2851,26.3198,0.0000
C00559=-38.969,-26.028,25.902,-150.1039,26.0381,0.0000
C00560=-41.068,-25.888,26.054,-149.7171,25.2803,0.0000
C00561=-43.046,-24.719,26.178,-149.2127,24.0648,0.0000
C00562=-44.510,-22.710,26.305,-148.7436,22.6029,0.0000
C00563=-45.665,-20.355,26.389,-148.3924,21.0774,0.0000
C00564=-46.683,-17.897,26.389,173.4316,36.8768,0.0000
C00565=-47.531,-15.415,26.305,175.1515,37.6247,0.0000
C00566=-47.917,-12.959,26.178,176.9251,38.2295,0.0000
C00567=-47.345,-10.734,26.054,178.4998,38.6376,0.0000
C00568=-45.960,-9.151,25.902,179.5392,38.8342,0.0000
C00569=-43.994,-8.395,25.615,179.9528,38.8795,0.0000
C00570=-41.862,-7.794,25.043,-179.7361,38.8953,0.0000
C00571=-39.979,-7.219,24.311,-179.4268,38.9091,0.0000
C00572=-38.594,-6.557,23.612,-179.0461,38.9341,0.0000
C00573=-37.838,-5.504,23.110,-178.4108,38.9797,0.0000
C00574=-37.737,-3.633,22.912,-177.2985,39.0231,0.0000
C00575=-37.849,-1.790,22.904,-177.2373,39.0582,0.0000
C00576=-37.892,0.000,22.909,-179.9995,39.1300,0.0000
C00577=-37.849,1.790,22.904,177.2375,39.0582,0.0000
C00578=-37.737,3.633,22.912,177.2991,39.0231,0.0000
C00579=-37.838,5.504,23.110,178.4114,38.9797,0.0000
C00580=-38.594,6.557,23.612,179.0467,38.9341,0.0000
C00581=-39.979,7.219,24.311,179.4273,38.9091,0.0000
C00582=-41.862,7.794,25.043,179.7367,38.8952,0.0000
C00583=-43.994,8.395,25.615,-179.9523,38.8795,0.0000
C00584=-45.960,9.151,25.902,-179.5386,38.8341,0.0000
C00585=-47.345,10.734,26.054,-178.4994,38.6375,0.0000
C00586=-47.917,12.959,26.178,-176.9249,38.2295,0.0000
C00587=-47.531,15.415,26.305,-175.1514,37.6246,0.0000
C00588=-46.683,17.897,26.389,-173.4316,36.8768,0.0000
C00589=-45.665,20.355,26.389,148.3924,21.0774,0.0000
C00590=-44.510,22.710,26.305,148.7436,22.6029,0.0000
C00591=-43.046,24.719,26.178,149.2128,24.0649,0.0000
C00592=-41.068,25.888,26.054,149.7173,25.2806,0.0000
C00593=-38.969,26.028,25.902,150.1041,26.0384,0.0000
C00594=-37.045,25.172,25.615,150.2853,26.3202,0.0000
C00595=-35.112,24.090,25.043,150.4374,26.5210,0.0000
C00596=-33.374,23.165,24.311,150.5899,26.7199,0.0000
C00597=-31.927,22.654,23.612,150.7702,26.9698,0.0000
C00598=-30.647,22.864,23.110,151.0666,27.3901,0.0000
C00599=-29.253,24.115,22.912,151.6154,28.1064,0.0000
C00600=-28.029,25.498,22.904,151.6159,28.1655,0.0000
C00601=-26.793,26.793,22.909,150.0900,26.5032,0.0000
C00602=-25.498,28.029,22.904,148.6761,24.7773,0.0000
C00603=-24.115,29.253,22.912,148.7393,24.7925,0.0000
C00604=-22.864,30.647,23.110,149.3737,25.4398,0.0000
C00605=-22.654,31.927,23.612,149.7534,25.7988,0.0000
C00606=-23.165,33.374,24.311,149.9788,26.0162,0.0000
C00607=-24.090,35.112,25.043,150.1562,26.1972,0.0000
C00608=-25.172,37.045,25.615,150.3361,26.3785,0.0000
C00609=-26.028,38.969,25.902,150.5967,26.6051,0.0000
C00610=-25.888,41.068,26.054,151.3255,27.1277,0.0000
C00611=-24.719,43.046,26.178,152.5326,27.8634,0.0000
C00612=-22.710,44.510,26.305,154.0336,28.6211,0.0000
C00613=-20.355,45.665,26.389,155.6510,29.2771,0.0000
C00614=-17.897,46.683,26.389,142.9419,-5.2501,0.0000
C00615=-15.415,47.531,26.305,142.2760,-3.8385,0.0000
C00616=-12.959,47.917,26.178,141.7304,-2.4152,0.0000
C00617=-10.734,47.345,26.054,141.3529,-1.1721,0.0000
C00618=-9.151,45.960,25.902,141.1650,-0.3594,0.0000
C00619=-8.395,43.994,25.615,141.1205,-0.0372,0.0000
C00620=-7.794,41.862,25.043,141.1045,0.2049,0.0000
C00621=-7.219,39.979,24.311,141.0895,0.4456,0.0000
C00622=-6.557,38.594,23.612,141.0621,0.7415,0.0000
C00623=-5.504,37.838,23.110,141.0096,1.2348,0.0000
C00624=-3.633,37.737,22.912,140.9457,2.0980,0.0000
C00625=-1.790,37.849,22.904,140.9092,2.1447,0.0000
C00626=0.000,37.892,22.909,140.8700,-0.0004,0.0000
C00627=0.000,36.499,24.612,141.0042,-0.0006,0.0000
C00628=1.663,36.461,24.606,141.0426,-2.1059,0.0000
C00629=3.419,36.362,24.616,141.0773,-2.0847,0.0000
C00630=5.241,36.506,24.842,141.1359,-1.2309,0.0000
C00631=6.234,37.375,25.413,141.1790,-0.7625,0.0000
C00632=6.845,38.939,26.213,141.1922,-0.4907,0.0000
C00633=7.384,41.061,27.051,141.1864,-0.2691,0.0000
C00634=7.952,43.467,27.704,141.1744,-0.0459,0.0000
C00635=8.667,45.697,28.032,141.1865,0.2540,0.0000
C00636=10.278,47.290,28.205,141.3530,1.0923,0.0000
C00637=12.598,47.983,28.348,141.7359,2.4182,0.0000
C00638=15.186,47.607,28.492,142.3234,3.9552,0.0000
C00639=17.819,46.713,28.587,143.0588,5.4819,0.0000
C00640=20.431,45.631,28.587,155.9249,-29.3784,0.0000
C00641=22.925,44.401,28.492,154.1600,-28.6808,0.0000
C00642=25.021,42.837,28.348,152.5396,-27.8622,0.0000
C00643=26.172,40.707,28.205,151.2701,-27.0651,0.0000
C00644=26.184,38.442,28.032,150.5431,-26.5088,0.0000
C00645=25.113,36.359,27.704,150.3265,-26.2798,0.0000
C00646=23.813,34.256,27.051,150.1844,-26.0963,0.0000
C00647=22.694,32.374,26.213,150.0383,-25.9176,0.0000
C00648=22.020,30.836,25.413,149.8419,-25.7107,0.0000
C00649=22.108,29.520,24.842,149.4872,-25.3661,0.0000
C00650=23.294,28.129,24.616,148.8634,-24.7235,0.0000
C00651=24.606,26.957,24.606,148.8189,-24.7276,0.0000
C00652=25.809,25.809,24.612,150.2077,-26.4201,0.0000
C00653=26.957,24.606,24.606,151.7064,-28.0518,0.0000
C00654=28.129,23.294,24.616,151.7219,-28.0133,0.0000
C00655=29.520,22.108,24.842,151.1748,-27.3080,0.0000
C00656=30.836,22.020,25.413,150.8874,-26.9134,0.0000
C00657=32.374,22.694,26.213,150.7110,-26.6914,0.0000
C00658=34.256,23.813,27.051,150.5531,-26.5204,0.0000
C00659=36.359,25.113,27.704,150.3892,-26.3519,0.0000
C00660=38.442,26.184,28.032,150.1946,-26.1078,0.0000
C00661=40.707,26.172,28.205,149.7710,-25.3431,0.0000
C00662=42.837,25.021,28.348,149.2154,-24.0588,0.0000
C00663=44.401,22.925,28.492,148.7078,-22.4813,0.0000
C00664=45.631,20.431,28.587,148.3415,-20.8224,0.0000
C00665=46.713,17.819,28.587,-173.1529,-36.7444,0.0000
C00666=47.607,15.186,28.492,-175.0075,-37.5713,0.0000
C00667=47.983,12.598,28.348,-176.9213,-38.2239,0.0000
C00668=47.290,10.278,28.205,-178.6015,-38.6387,0.0000
C00669=45.697,8.667,28.032,-179.6741,-38.8131,0.0000
C00670=43.467,7.952,27.704,179.9410,-38.8256,0.0000
C00671=41.061,7.384,27.051,179.6547,-38.8131,0.0000
C00672=38.939,6.845,26.213,179.3703,-38.8061,0.0000
C00673=37.375,6.234,25.413,179.0213,-38.8169,0.0000
C00674=36.506,5.241,24.842,178.4193,-38.8535,0.0000
C00675=36.362,3.419,24.616,177.3212,-38.8921,0.0000
C00676=36.461,1.663,24.606,177.2927,-38.9261,0.0000
C00677=36.499,0.000,24.612,179.9992,-38.9958,0.0000
C00678=36.461,-1.662,24.606,-177.2929,-38.9262,0.0000
C00679=36.362,-3.419,24.616,-177.3219,-38.8921,0.0000
C00680=36.506,-5.241,24.842,-178.4199,-38.8534,0.0000
C00681=37.375,-6.234,25.413,-179.0219,-38.8169,0.0000
C00682=38.939,-6.845,26.213,-179.3708,-38.8061,0.0000
C00683=41.061,-7.384,27.051,-179.6552,-38.8131,0.0000
C00684=43.467,-7.952,27.704,-179.9416,-38.8256,0.0000
C00685=45.697,-8.667,28.032,179.6736,-38.8130,0.0000
C00686=47.290,-10.278,28.205,178.6011,-38.6386,0.0000
C00687=47.983,-12.598,28.348,176.9211,-38.2238,0.0000
C00688=47.607,-15.186,28.492,175.0074,-37.5712,0.0000
C00689=46.713,-17.819,28.587,173.1529,-36.7444,0.0000
C00690=45.631,-20.431,28.587,-148.3415,-20.8224,0.0000
C00691=44.401,-22.925,28.492,-148.7078,-22.4814,0.0000
C00692=42.837,-25.021,28.348,-149.2155,-24.0590,0.0000
C00693=40.707,-26.172,28.205,-149.7711,-25.3434,0.0000
C00694=38.442,-26.184,28.032,-150.1948,-26.1082,0.0000
C00695=36.359,-25.113,27.704,-150.3895,-26.3523,0.0000
C00696=34.256,-23.813,27.051,-150.5534,-26.5208,0.0000
C00697=32.374,-22.694,26.213,-150.7113,-26.6918,0.0000
C00698=30.836,-22.020,25.413,-150.8876,-26.9138,0.0000
C00699=29.520,-22.108,24.842,-151.1751,-27.3084,0.0000
C00700=28.129,-23.294,24.616,-151.7223,-28.0137,0.0000
C00701=26.957,-24.606,24.606,-151.7065,-28.0519,0.0000
C00702=25.809,-25.809,24.612,-150.2085,-26.4210,0.0000
C00703=24.606,-26.957,24.606,-148.8189,-24.7278,0.0000
C00704=23.294,-28.129,24.616,-148.8638,-24.7239,0.0000
C00705=22.108,-29.520,24.842,-149.4876,-25.3664,0.0000
C00706=22.020,-30.836,25.413,-149.8423,-25.7111,0.0000
C00707=22.694,-32.374,26.213,-150.0387,-25.9179,0.0000
C00708=23.813,-34.256,27.051,-150.1848,-26.0966,0.0000
C00709=25.113,-36.359,27.704,-150.3268,-26.2801,0.0000
C00710=26.184,-38.442,28.032,-150.5434,-26.5091,0.0000
C00711=26.172,-40.707,28.205,-151.2703,-27.0653,0.0000
C00712=25.021,-42.837,28.348,-152.5398,-27.8623,0.0000
C00713=22.925,-44.401,28.492,-154.1600,-28.6809,0.0000
C00714=20.431,-45.631,28.587,-155.9249,-29.3784,0.0000
C00715=17.819,-46.713,28.587,-143.0588,5.4819,0.0000
C00716=15.186,-47.607,28.492,-142.3234,3.9552,0.0000
C00717=12.598,-47.983,28.348,-141.7359,2.4182,0.0000
C00718=10.278,-47.290,28.205,-141.3530,1.0923,0.0000
C00719=8.667,-45.697,28.032,-141.1865,0.2540,0.0000
C00720=7.952,-43.467,27.704,-141.1744,-0.0459,0.0000
C00721=7.384,-41.061,27.051,-141.1864,-0.2691,0.0000
C00722=6.845,-38.939,26.213,-141.1922,-0.4907,0.0000
C00723=6.234,-37.375,25.413,-141.1790,-0.7625,0.0000
C00724=5.241,-36.506,24.842,-141.1359,-1.2309,0.0000
C00725=3.419,-36.362,24.616,-141.0773,-2.0847,0.0000
C00726=1.663,-36.461,24.606,-141.0426,-2.1059,0.0000
C00727=0.000,-36.499,24.612,-141.0042,-0.0006,0.0000
C00728=0.000,-36.499,24.612,-141.0042,-0.0006,0.0000
C00729=-1.662,-36.461,24.606,-141.0425,2.1057,0.0000
C00730=-3.419,-36.362,24.616,-141.0773,2.0841,0.0000
C00731=-5.241,-36.506,24.842,-141.1359,1.2304,0.0000
C00732=-6.234,-37.375,25.413,-141.1790,0.7621,0.0000
C00733=-6.845,-38.939,26.213,-141.1923,0.4903,0.0000
C00734=-7.384,-41.061,27.051,-141.1864,0.2686,0.0000
C00735=-7.952,-43.467,27.704,-141.1744,0.0455,0.0000
C00736=-8.667,-45.697,28.032,-141.1866,-0.2544,0.0000
C00737=-10.278,-47.290,28.205,-141.3531,-1.0926,0.0000
C00738=-12.598,-47.983,28.348,-141.7359,-2.4184,0.0000
C00739=-15.186,-47.607,28.492,-142.3235,-3.9553,0.0000
C00740=-17.819,-46.713,28.587,-143.0588,-5.4819,0.0000
C00741=-20.431,-45.631,28.587,-155.9249,29.3784,0.0000
C00742=-22.925,-44.401,28.492,-154.1600,28.6808,0.0000
C00743=-25.021,-42.837,28.348,-152.5396,27.8622,0.0000
C00744=-26.172,-40.707,28.205,-151.2701,27.0651,0.0000
C00745=-26.184,-38.442,28.032,-150.5431,26.5088,0.0000
C00746=-25.113,-36.359,27.704,-150.3265,26.2798,0.0000
C00747=-23.813,-34.256,27.051,-150.1844,26.0963,0.0000
C00748=-22.694,-32.374,26.213,-150.0383,25.9176,0.0000
C00749=-22.020,-30.836,25.413,-149.8419,25.7107,0.0000
C00750=-22.108,-29.520,24.842,-149.4872,25.3661,0.0000
C00751=-23.294,-28.129,24.616,-148.8634,24.7235,0.0000
C00752=-24.606,-26.957,24.606,-148.8189,24.7276,0.0000
C00753=-25.809,-25.809,24.612,-150.2077,26.4201,0.0000
C00754=-26.957,-24.606,24.606,-151.7064,28.0518,0.0000
C00755=-28.129,-23.294,24.616,-151.7219,28.0133,0.0000
C00756=-29.520,-22.108,24.842,-151.1748,27.3080,0.0000
C00757=-30.836,-22.020,25.413,-150.8874,26.9134,0.0000
C00758=-32.374,-22.694,26.213,-150.7110,26.6914,0.0000
C00759=-34.256,-23.813,27.051,-150.5531,26.5204,0.0000
C00760=-36.359,-25.113,27.704,-150.3892,26.3519,0.0000
C00761=-38.442,-26.184,28.032,-150.1946,26.1078,0.0000
C00762=-40.707,-26.172,28.205,-149.7710,25.3431,0.0000
C00763=-42.837,-25.021,28.348,-149.2154,24.0589,0.0000
C00764=-44.401,-22.925,28.492,-148.7078,22.4813,0.0000
C00765=-45.631,-20.431,28.587,-148.3415,20.8224,0.0000
C00766=-46.713,-17.819,28.587,173.1529,36.7444,0.0000
C00767=-47.607,-15.186,28.492,175.0075,37.5713,0.0000
C00768=-47.983,-12.598,28.348,176.9213,38.2239,0.0000
C00769=-47.290,-10.278,28.205,178.6015,38.6387,0.0000
C00770=-45.697,-8.667,28.032,179.6741,38.8131,0.0000
C00771=-43.467,-7.952,27.704,-179.9410,38.8256,0.0000
C00772=-41.061,-7.384,27.051,-179.6547,38.8131,0.0000
C00773=-38.939,-6.845,26.213,-179.3703,38.8061,0.0000
C00774=-37.375,-6.234,25.413,-179.0213,38.8169,0.0000
C00775=-36.506,-5.241,24.842,-178.4193,38.8535,0.0000
C00776=-36.362,-3.419,24.616,-177.3212,38.8921,0.0000
C00777=-36.461,-1.663,24.606,-177.2927,38.9261,0.0000
C00778=-36.499,0.000,24.612,-179.9992,38.9958,0.0000
C00779=-36.461,1.662,24.606,177.2929,38.9262,0.0000
C00780=-36.362,3.419,24.616,177.3219,38.8921,0.0000
C00781=-36.506,5.241,24.842,178.4199,38.8534,0.0000
C00782=-37.375,6.234,25.413,179.0219,38.8169,0.0000
C00783=-38.939,6.845,26.213,179.3708,38.8061,0.0000
C00784=-41.061,7.384,27.051,179.6552,38.8131,0.0000
C00785=-43.467,7.952,27.704,179.9416,38.8256,0.0000
C00786=-45.697,8.667,28.032,-179.6736,38.8130,0.0000
C00787=-47.290,10.278,28.205,-178.6011,38.6386,0.0000
C00788=-47.983,12.598,28.348,-176.9211,38.2238,0.0000
C00789=-47.607,15.186,28.492,-175.0074,37.5712,0.0000
C00790=-46.713,17.819,28.587,-173.1529,36.7444,0.0000
C00791=-45.631,20.431,28.587,148.3415,20.8224,0.0000
C00792=-44.401,22.925,28.492,148.7078,22.4814,0.0000
C00793=-42.837,25.021,28.348,149.2155,24.0590,0.0000
C00794=-40.707,26.172,28.205,149.7711,25.3434,0.0000
C00795=-38.442,26.184,28.032,150.1948,26.1082,0.0000
C00796=-36.359,25.113,27.704,150.3895,26.3523,0.0000
C00797=-34.256,23.813,27.051,150.5534,26.5208,0.0000
C00798=-32.374,22.694,26.213,150.7113,26.6918,0.0000
C00799=-30.836,22.020,25.413,150.8876,26.9138,0.0000
C00800=-29.520,22.108,24.842,151.1751,27.3084,0.0000
C00801=-28.129,23.294,24.616,151.7223,28.0137,0.0000
C00802=-26.957,24.606,24.606,151.7065,28.0519,0.0000
C00803=-25.809,25.809,24.612,150.2085,26.4210,0.0000
C00804=-24.606,26.957,24.606,148.8189,24.7278,0.0000
C00805=-23.294,28.129,24.616,148.8638,24.7239,0.0000
C00806=-22.108,29.520,24.842,149.4876,25.3664,0.0000
C00807=-22.020,30.836,25.413,149.8423,25.7111,0.0000
C00808=-22.694,32.374,26.213,150.0387,25.9179,0.0000
C00809=-23.813,34.256,27.051,150.1848,26.0966,0.0000
C00810=-25.113,36.359,27.704,150.3268,26.2801,0.0000
C00811=-26.184,38.442,28.032,150.5434,26.5091,0.0000
C00812=-26.172,40.707,28.205,151.2703,27.0653,0.0000
C00813=-25.021,42.837,28.348,152.5398,27.8623,0.0000
C00814=-22.925,44.401,28.492,154.1600,28.6809,0.0000
C00815=-20.431,45.631,28.587,155.9249,29.3784,0.0000
C00816=-17.819,46.713,28.587,143.0588,-5.4819,0.0000
C00817=-15.186,47.607,28.492,142.3235,-3.9553,0.0000
C00818=-12.598,47.983,28.348,141.7359,-2.4184,0.0000
C00819=-10.278,47.290,28.205,141.3531,-1.0926,0.0000
C00820=-8.667,45.697,28.032,141.1866,-0.2544,0.0000
C00821=-7.952,43.467,27.704,141.1744,0.0455,0.0000
C00822=-7.384,41.061,27.051,141.1864,0.2686,0.0000
C00823=-6.845,38.939,26.213,141.1923,0.4903,0.0000
C00824=-6.234,37.375,25.413,141.1790,0.7621,0.0000
C00825=-5.241,36.506,24.842,141.1359,1.2304,0.0000
C00826=-3.419,36.362,24.616,141.0773,2.0841,0.0000
C00827=-1.662,36.461,24.606,141.0425,2.1057,0.0000
C00828=0.000,36.499,24.612,141.0042,-0.0006,0.0000
C00829=0.000,35.110,26.318,141.1763,-0.0008,0.0000
C00830=1.536,35.076,26.311,141.2137,-2.0625,0.0000
C00831=3.206,34.989,26.322,141.2468,-2.0729,0.0000
C00832=4.979,35.179,26.576,141.3004,-1.2312,0.0000
C00833=5.912,36.162,27.221,141.3343,-0.7891,0.0000
C00834=6.475,37.910,28.122,141.3331,-0.5417,0.0000
C00835=6.981,40.274,29.065,141.3055,-0.3387,0.0000
C00836=7.520,42.952,29.799,141.2634,-0.1338,0.0000
C00837=8.198,45.442,30.166,141.2406,0.1443,0.0000
C00838=9.836,47.237,30.360,141.3828,1.0101,0.0000
C00839=12.248,48.046,30.519,141.7693,2.4203,0.0000
C00840=14.965,47.679,30.679,142.3999,4.0724,0.0000
C00841=17.744,46.742,30.786,143.2079,5.7137,0.0000
C00842=20.505,45.599,30.786,156.2273,-29.4583,0.0000
C00843=23.132,44.297,30.679,154.3122,-28.7224,0.0000
C00844=25.313,42.634,30.519,152.5705,-27.8429,0.0000
C00845=26.446,40.357,30.360,151.2390,-26.9821,0.0000
C00846=26.335,37.929,30.166,150.5153,-26.3891,0.0000
C00847=25.054,35.689,29.799,150.3446,-26.1558,0.0000
C00848=23.542,33.414,29.065,150.2415,-25.9683,0.0000
C00849=22.228,31.385,28.122,150.1273,-25.7909,0.0000
C00850=21.390,29.751,27.221,149.9602,-25.5947,0.0000
C00851=21.354,28.396,26.576,149.6312,-25.2655,0.0000
C00852=22.474,27.008,26.322,149.0195,-24.6301,0.0000
C00853=23.717,25.889,26.311,148.9976,-24.6585,0.0000
C00854=24.826,24.826,26.318,150.3591,-26.3142,0.0000
C00855=25.888,23.717,26.311,151.8272,-27.9113,0.0000
C00856=27.008,22.474,26.322,151.8636,-27.8985,0.0000
C00857=28.396,21.354,26.576,151.3202,-27.2063,0.0000
C00858=29.751,21.390,27.221,151.0427,-26.8383,0.0000
C00859=31.385,22.228,28.122,150.8703,-26.6446,0.0000
C00860=33.414,23.542,29.065,150.7059,-26.5018,0.0000
C00861=35.689,25.054,29.799,150.5279,-26.3664,0.0000
C00862=37.929,26.335,30.166,150.3172,-26.1611,0.0000
C00863=40.357,26.446,30.360,149.8527,-25.3900,0.0000
C00864=42.634,25.313,30.519,149.2430,-24.0369,0.0000
C00865=44.297,23.132,30.679,148.6966,-22.3418,0.0000
C00866=45.599,20.505,30.786,148.3180,-20.5481,0.0000
C00867=46.742,17.744,30.786,-172.8783,-36.5795,0.0000
C00868=47.679,14.965,30.679,-174.8650,-37.4888,0.0000
C00869=48.046,12.248,30.519,-176.9201,-38.1905,0.0000
C00870=47.237,9.836,30.360,-178.7073,-38.6101,0.0000
C00871=45.442,8.198,30.166,-179.8150,-38.7592,0.0000
C00872=42.952,7.520,29.799,179.8284,-38.7365,0.0000
C00873=40.274,6.981,29.065,179.5661,-38.6937,0.0000
C00874=37.910,6.475,28.122,179.3062,-38.6648,0.0000
C00875=36.162,5.912,27.221,178.9894,-38.6613,0.0000
C00876=35.179,4.979,26.576,178.4226,-38.6890,0.0000
C00877=34.989,3.206,26.322,177.3426,-38.7231,0.0000
C00878=35.076,1.536,26.311,177.3548,-38.7565,0.0000
C00879=35.110,0.000,26.318,179.9990,-38.8237,0.0000
C00880=35.076,-1.535,26.311,-177.3549,-38.7565,0.0000
C00881=34.989,-3.206,26.322,-177.3434,-38.7231,0.0000
C00882=35.179,-4.979,26.576,-178.4232,-38.6890,0.0000
C00883=36.162,-5.912,27.221,-178.9899,-38.6613,0.0000
C00884=37.910,-6.475,28.122,-179.3067,-38.6648,0.0000
C00885=40.274,-6.981,29.065,-179.5666,-38.6937,0.0000
C00886=42.952,-7.520,29.799,-179.8290,-38.7364,0.0000
C00887=45.442,-8.198,30.166,179.8144,-38.7592,0.0000
C00888=47.237,-9.836,30.360,178.7069,-38.6101,0.0000
C00889=48.046,-12.248,30.519,176.9198,-38.1904,0.0000
C00890=47.679,-14.965,30.679,174.8649,-37.4887,0.0000
C00891=46.742,-17.744,30.786,172.8783,-36.5795,0.0000
C00892=45.599,-20.505,30.786,-148.3180,-20.5481,0.0000
C00893=44.297,-23.132,30.679,-148.6966,-22.3419,0.0000
C00894=42.634,-25.313,30.519,-149.2431,-24.0371,0.0000
C00895=40.357,-26.446,30.360,-149.8528,-25.3903,0.0000
C00896=37.929,-26.335,30.166,-150.3174,-26.1615,0.0000
C00897=35.689,-25.054,29.799,-150.5281,-26.3668,0.0000
C00898=33.414,-23.542,29.065,-150.7061,-26.5022,0.0000
C00899=31.385,-22.228,28.122,-150.8706,-26.6449,0.0000
C00900=29.751,-21.390,27.221,-151.0429,-26.8386,0.0000
C00901=28.396,-21.354,26.576,-151.3205,-27.2067,0.0000
C00902=27.008,-22.474,26.322,-151.8640,-27.8989,0.0000
C00903=25.889,-23.717,26.311,-151.8273,-27.9114,0.0000
C00904=24.826,-24.826,26.318,-150.3602,-26.3155,0.0000
C00905=23.717,-25.888,26.311,-148.9976,-24.6586,0.0000
C00906=22.474,-27.008,26.322,-149.0199,-24.6306,0.0000
C00907=21.354,-28.396,26.576,-149.6315,-25.2659,0.0000
C00908=21.390,-29.751,27.221,-149.9605,-25.5950,0.0000
C00909=22.228,-31.385,28.122,-150.1277,-25.7913,0.0000
C00910=23.542,-33.414,29.065,-150.2419,-25.9686,0.0000
C00911=25.054,-35.689,29.799,-150.3449,-26.1561,0.0000
C00912=26.335,-37.929,30.166,-150.5157,-26.3894,0.0000
C00913=26.446,-40.357,30.360,-151.2393,-26.9823,0.0000
C00914=25.313,-42.634,30.519,-152.5706,-27.8430,0.0000
C00915=23.132,-44.297,30.679,-154.3123,-28.7225,0.0000
C00916=20.505,-45.599,30.786,-156.2273,-29.4583,0.0000
C00917=17.744,-46.742,30.786,-143.2079,5.7137,0.0000
C00918=14.965,-47.679,30.679,-142.3999,4.0724,0.0000
C00919=12.248,-48.046,30.519,-141.7693,2.4203,0.0000
C00920=9.836,-47.237,30.360,-141.3828,1.0101,0.0000
C00921=8.198,-45.442,30.166,-141.2406,0.1443,0.0000
C00922=7.520,-42.952,29.799,-141.2634,-0.1338,0.0000
C00923=6.981,-40.274,29.065,-141.3055,-0.3387,0.0000
C00924=6.475,-37.910,28.122,-141.3331,-0.5417,0.0000
C00925=5.912,-36.162,27.221,-141.3343,-0.7891,0.0000
C00926=4.979,-35.179,26.576,-141.3004,-1.2312,0.0000
C00927=3.206,-34.989,26.322,-141.2468,-2.0729,0.0000
C00928=1.536,-35.076,26.311,-141.2137,-2.0625,0.0000
C00929=0.000,-35.110,26.318,-141.1763,-0.0008,0.0000
C00930=0.000,-35.110,26.318,-141.1763,-0.0008,0.0000
C00931=-1.535,-35.076,26.311,-141.2136,2.0624,0.0000
C00932=-3.206,-34.989,26.322,-141.2468,2.0724,0.0000
C00933=-4.979,-35.179,26.576,-141.3004,1.2307,0.0000
C00934=-5.912,-36.162,27.221,-141.3344,0.7887,0.0000
C00935=-6.475,-37.910,28.122,-141.3332,0.5413,0.0000
C00936=-6.981,-40.274,29.065,-141.3055,0.3382,0.0000
C00937=-7.520,-42.952,29.799,-141.2634,0.1334,0.0000
C00938=-8.198,-45.442,30.166,-141.2407,-0.1447,0.0000
C00939=-9.836,-47.237,30.360,-141.3828,-1.0104,0.0000
C00940=-12.248,-48.046,30.519,-141.7693,-2.4205,0.0000
C00941=-14.965,-47.679,30.679,-142.3999,-4.0725,0.0000
C00942=-17.744,-46.742,30.786,-143.2079,-5.7137,0.0000
C00943=-20.505,-45.599,30.786,-156.2273,29.4583,0.0000
C00944=-23.132,-44.297,30.679,-154.3122,28.7224,0.0000
C00945=-25.313,-42.634,30.519,-152.5705,27.8429,0.0000
C00946=-26.446,-40.357,30.360,-151.2390,26.9821,0.0000
C00947=-26.335,-37.929,30.166,-150.5153,26.3891,0.0000
C00948=-25.054,-35.689,29.799,-150.3446,26.1558,0.0000
C00949=-23.542,-33.414,29.065,-150.2415,25.9683,0.0000
C00950=-22.228,-31.385,28.122,-150.1273,25.7909,0.0000
C00951=-21.390,-29.751,27.221,-149.9602,25.5947,0.0000
C00952=-21.354,-28.396,26.576,-149.6312,25.2655,0.0000
C00953=-22.474,-27.008,26.322,-149.0195,24.6301,0.0000
C00954=-23.717,-25.889,26.311,-148.9976,24.6585,0.0000
C00955=-24.826,-24.826,26.318,-150.3591,26.3142,0.0000
C00956=-25.888,-23.717,26.311,-151.8272,27.9113,0.0000
C00957=-27.008,-22.474,26.322,-151.8636,27.8985,0.0000
C00958=-28.396,-21.354,26.576,-151.3202,27.2063,0.0000
C00959=-29.751,-21.390,27.221,-151.0427,26.8383,0.0000
C00960=-31.385,-22.228,28.122,-150.8703,26.6446,0.0000
C00961=-33.414,-23.542,29.065,-150.7059,26.5018,0.0000
C00962=-35.689,-25.054,29.799,-150.5279,26.3664,0.0000
C00963=-37.929,-26.335,30.166,-150.3172,26.1611,0.0000
C00964=-40.357,-26.446,30.360,-149.8527,25.3900,0.0000
C00965=-42.634,-25.313,30.519,-149.2430,24.0369,0.0000
C00966=-44.297,-23.132,30.679,-148.6966,22.3418,0.0000
C00967=-45.599,-20.505,30.786,-148.3180,20.5481,0.0000
C00968=-46.742,-17.744,30.786,172.8783,36.5795,0.0000
C00969=-47.679,-14.965,30.679,174.8650,37.4888,0.0000
C00970=-48.046,-12.248,30.519,176.9201,38.1905,0.0000
C00971=-47.237,-9.836,30.360,178.7073,38.6101,0.0000
C00972=-45.442,-8.198,30.166,179.8150,38.7592,0.0000
C00973=-42.952,-7.520,29.799,-179.8284,38.7365,0.0000
C00974=-40.274,-6.981,29.065,-179.5661,38.6937,0.0000
C00975=-37.910,-6.475,28.122,-179.3062,38.6648,0.0000
C00976=-36.162,-5.912,27.221,-178.9894,38.6613,0.0000
C00977=-35.179,-4.979,26.576,-178.4226,38.6890,0.0000
C00978=-34.989,-3.206,26.322,-177.3426,38.7231,0.0000
C00979=-35.076,-1.536,26.311,-177.3548,38.7565,0.0000
C00980=-35.110,0.000,26.318,-179.9990,38.8237,0.0000
C00981=-35.076,1.535,26.311,177.3549,38.7565,0.0000
C00982=-34.989,3.206,26.322,177.3434,38.7231,0.0000
C00983=-35.179,4.979,26.576,178.4232,38.6890,0.0000
C00984=-36.162,5.912,27.221,178.9899,38.6613,0.0000
C00985=-37.910,6.475,28.122,179.3067,38.6648,0.0000
C00986=-40.274,6.981,29.065,179.5666,38.6937,0.0000
C00987=-42.952,7.520,29.799,179.8290,38.7364,0.0000
C00988=-45.442,8.198,30.166,-179.8144,38.7592,0.0000
C00989=-47.237,9.836,30.360,-178.7069,38.6101,0.0000
C00990=-48.046,12.248,30.519,-176.9198,38.1904,0.0000
C00991=-47.679,14.965,30.679,-174.8649,37.4887,0.0000
C00992=-46.742,17.744,30.786,-172.8783,36.5795,0.0000
C00993=-45.599,20.505,30.786,148.3180,20.5481,0.0000
C00994=-44.297,23.132,30.679,148.6966,22.3419,0.0000
C00995=-42.634,25.313,30.519,149.2431,24.0371,0.0000
C00996=-40.357,26.446,30.360,149.8528,25.3903,0.0000
C00997=-37.929,26.335,30.166,150.3174,26.1615,0.0000
C00998=-35.689,25.054,29.799,150.5281,26.3668,0.0000
C00999=-33.414,23.542,29.065,150.7061,26.5022,0.0000
C01000=-31.385,22.228,28.122,150.8706,26.6449,0.0000
C01001=-29.751,21.390,27.221,151.0429,26.8386,0.0000
C01002=-28.396,21.354,26.576,151.3205,27.2067,0.0000
C01003=-27.008,22.474,26.322,151.8640,27.8989,0.0000
C01004=-25.889,23.717,26.311,151.8273,27.9114,0.0000
C01005=-24.826,24.826,26.318,150.3602,26.3155,0.0000
C01006=-23.717,25.888,26.311,148.9976,24.6586,0.0000
C01007=-22.474,27.008,26.322,149.0199,24.6306,0.0000
C01008=-21.354,28.396,26.576,149.6315,25.2659,0.0000
C01009=-21.390,29.751,27.221,149.9605,25.5950,0.0000
C01010=-22.228,31.385,28.122,150.1277,25.7913,0.0000
C01011=-23.542,33.414,29.065,150.2419,25.9686,0.0000
C01012=-25.054,35.689,29.799,150.3449,26.1561,0.0000
C01013=-26.335,37.929,30.166,150.5157,26.3894,0.0000
C01014=-26.446,40.357,30.360,151.2393,26.9823,0.0000
C01015=-25.313,42.634,30.519,152.5706,27.8430,0.0000
C01016=-23.132,44.297,30.679,154.3123,28.7225,0.0000
C01017=-20.505,45.599,30.786,156.2273,29.4583,0.0000
C01018=-17.744,46.742,30.786,143.2079,-5.7137,0.0000
C01019=-14.965,47.679,30.679,142.3999,-4.0725,0.0000
C01020=-12.248,48.046,30.519,141.7693,-2.4205,0.0000
C01021=-9.836,47.237,30.360,141.3828,-1.0104,0.0000
C01022=-8.198,45.442,30.166,141.2407,-0.1447,0.0000
C01023=-7.520,42.952,29.799,141.2634,0.1334,0.0000
C01024=-6.981,40.274,29.065,141.3055,0.3382,0.0000
C01025=-6.475,37.910,28.122,141.3332,0.5413,0.0000
C01026=-5.912,36.162,27.221,141.3344,0.7887,0.0000
C01027=-4.979,35.179,26.576,141.3004,1.2307,0.0000
C01028=-3.206,34.989,26.322,141.2468,2.0724,0.0000
C01029=-1.535,35.076,26.311,141.2136,2.0624,0.0000
C01030=0.000,35.110,26.318,141.1763,-0.0008,0.0000
C01031=0.000,33.732,28.034,141.3848,-0.0010,0.0000
C01032=1.410,33.704,28.025,141.4210,-2.0148,0.0000
C01033=2.994,33.629,28.038,141.4528,-2.0626,0.0000
C01034=4.720,33.865,28.321,141.5015,-1.2352,0.0000
C01035=5.595,34.967,29.040,141.5266,-0.8200,0.0000
C01036=6.113,36.903,30.045,141.5109,-0.5966,0.0000
C01037=6.591,39.512,31.092,141.4604,-0.4109,0.0000
C01038=7.106,42.459,31.903,141.3865,-0.2227,0.0000
C01039=7.750,45.198,32.306,141.3268,0.0349,0.0000
C01040=9.416,47.186,32.519,141.4422,0.9302,0.0000
C01041=11.916,48.107,32.693,141.8310,2.4257,0.0000
C01042=14.756,47.748,32.868,142.5059,4.1932,0.0000
C01043=17.673,46.769,32.984,143.3894,5.9463,0.0000
C01044=20.574,45.568,32.984,156.5587,-29.5172,0.0000
C01045=23.329,44.198,32.868,154.4930,-28.7476,0.0000
C01046=25.591,42.442,32.693,152.6285,-27.8084,0.0000
C01047=26.708,40.024,32.519,151.2358,-26.8826,0.0000
C01048=26.480,37.440,32.306,150.5160,-26.2498,0.0000
C01049=24.998,35.047,31.903,150.3919,-26.0100,0.0000
C01050=23.279,32.600,31.092,150.3282,-25.8161,0.0000
C01051=21.772,30.417,30.045,150.2457,-25.6386,0.0000
C01052=20.769,28.682,29.040,150.1076,-25.4525,0.0000
C01053=20.608,27.283,28.321,149.8045,-25.1396,0.0000
C01054=21.662,25.896,28.038,149.2062,-24.5133,0.0000
C01055=22.835,24.829,28.025,149.2105,-24.5706,0.0000
C01056=23.852,23.852,28.034,150.5423,-26.1858,0.0000
C01057=24.829,22.835,28.025,151.9767,-27.7448,0.0000
C01058=25.896,21.662,28.038,152.0381,-27.7619,0.0000
C01059=27.283,20.608,28.321,151.5000,-27.0845,0.0000
C01060=28.682,20.769,29.040,151.2332,-26.7435,0.0000
C01061=30.417,21.772,30.045,151.0645,-26.5778,0.0000
C01062=32.600,23.279,31.092,150.8918,-26.4630,0.0000
C01063=35.047,24.998,31.903,150.6972,-26.3606,0.0000
C01064=37.440,26.480,32.306,150.4678,-26.1944,0.0000
C01065=40.024,26.708,32.519,149.9588,-25.4168,0.0000
C01066=42.442,25.591,32.693,149.2929,-23.9951,0.0000
C01067=44.198,23.329,32.868,148.7084,-22.1817,0.0000
C01068=45.568,20.574,32.984,148.3213,-20.2537,0.0000
C01069=46.769,17.673,32.984,-172.6068,-36.3819,0.0000
C01070=47.748,14.756,32.868,-174.7206,-37.3765,0.0000
C01071=48.107,11.916,32.693,-176.9157,-38.1287,0.0000
C01072=47.186,9.416,32.519,-178.8105,-38.5518,0.0000
C01073=45.198,7.750,32.306,-179.9553,-38.6732,0.0000
C01074=42.459,7.106,31.903,179.7150,-38.6132,0.0000
C01075=39.512,6.591,31.092,179.4747,-38.5384,0.0000
C01076=36.903,6.113,30.045,179.2379,-38.4867,0.0000
C01077=34.967,5.595,29.040,178.9526,-38.4687,0.0000
C01078=33.865,4.720,28.321,178.4219,-38.4879,0.0000
C01079=33.629,2.994,28.038,177.3634,-38.5176,0.0000
C01080=33.704,1.410,28.025,177.4234,-38.5507,0.0000
C01081=33.732,0.000,28.034,179.9987,-38.6152,0.0000
C01082=33.704,-1.410,28.025,-177.4234,-38.5508,0.0000
C01083=33.629,-2.994,28.038,-177.3641,-38.5176,0.0000
C01084=33.865,-4.720,28.321,-178.4225,-38.4879,0.0000
C01085=34.967,-5.595,29.040,-178.9532,-38.4687,0.0000
C01086=36.903,-6.113,30.045,-179.2384,-38.4866,0.0000
C01087=39.512,-6.591,31.092,-179.4753,-38.5384,0.0000
C01088=42.459,-7.106,31.903,-179.7156,-38.6131,0.0000
C01089=45.198,-7.750,32.306,179.9547,-38.6732,0.0000
C01090=47.186,-9.416,32.519,178.8100,-38.5517,0.0000
C01091=48.107,-11.916,32.693,176.9155,-38.1287,0.0000
C01092=47.748,-14.756,32.868,174.7205,-37.3765,0.0000
C01093=46.769,-17.673,32.984,172.6067,-36.3819,0.0000
C01094=45.568,-20.574,32.984,-148.3213,-20.2537,0.0000
C01095=44.198,-23.329,32.868,-148.7085,-22.1818,0.0000
C01096=42.442,-25.591,32.693,-149.2930,-23.9953,0.0000
C01097=40.024,-26.708,32.519,-149.9590,-25.4171,0.0000
C01098=37.440,-26.480,32.306,-150.4681,-26.1948,0.0000
C01099=35.047,-24.998,31.903,-150.6974,-26.3609,0.0000
C01100=32.600,-23.279,31.092,-150.8921,-26.4634,0.0000
C01101=30.417,-21.772,30.045,-151.0648,-26.5781,0.0000
C01102=28.682,-20.769,29.040,-151.2334,-26.7438,0.0000
C01103=27.283,-20.608,28.321,-151.5004,-27.0849,0.0000
C01104=25.896,-21.662,28.038,-152.0385,-27.7623,0.0000
C01105=24.829,-22.835,28.025,-151.9767,-27.7448,0.0000
C01106=23.852,-23.852,28.034,-150.5437,-26.1874,0.0000
C01107=22.835,-24.829,28.025,-149.2105,-24.5706,0.0000
C01108=21.662,-25.896,28.038,-149.2066,-24.5137,0.0000
C01109=20.608,-27.283,28.321,-149.8048,-25.1400,0.0000
C01110=20.769,-28.682,29.040,-150.1079,-25.4528,0.0000
C01111=21.772,-30.417,30.045,-150.2461,-25.6389,0.0000
C01112=23.279,-32.600,31.092,-150.3285,-25.8165,0.0000
C01113=24.998,-35.047,31.903,-150.3922,-26.0104,0.0000
C01114=26.480,-37.440,32.306,-150.5163,-26.2501,0.0000
C01115=26.708,-40.024,32.519,-151.2361,-26.8828,0.0000
C01116=25.591,-42.442,32.693,-152.6287,-27.8086,0.0000
C01117=23.329,-44.198,32.868,-154.4930,-28.7477,0.0000
C01118=20.574,-45.568,32.984,-156.5587,-29.5172,0.0000
C01119=17.673,-46.769,32.984,-143.3894,5.9463,0.0000
C01120=14.756,-47.748,32.868,-142.5059,4.1932,0.0000
C01121=11.916,-48.107,32.693,-141.8310,2.4257,0.0000
C01122=9.416,-47.186,32.519,-141.4422,0.9302,0.0000
C01123=7.750,-45.198,32.306,-141.3268,0.0349,0.0000
C01124=7.106,-42.459,31.903,-141.3865,-0.2227,0.0000
C01125=6.591,-39.512,31.092,-141.4604,-0.4109,0.0000
C01126=6.113,-36.903,30.045,-141.5109,-0.5966,0.0000
C01127=5.595,-34.967,29.040,-141.5266,-0.8200,0.0000
C01128=4.720,-33.865,28.321,-141.5015,-1.2352,0.0000
C01129=2.994,-33.629,28.038,-141.4528,-2.0626,0.0000
C01130=1.410,-33.704,28.025,-141.4210,-2.0148,0.0000
C01131=0.000,-33.732,28.034,-141.3848,-0.0010,0.0000
C01132=0.000,-33.732,28.034,-141.3848,-0.0010,0.0000
C01133=-1.410,-33.704,28.025,-141.4210,2.0148,0.0000
C01134=-2.994,-33.629,28.038,-141.4528,2.0621,0.0000
C01135=-4.720,-33.865,28.321,-141.5015,1.2347,0.0000
C01136=-5.595,-34.967,29.040,-141.5266,0.8196,0.0000
C01137=-6.113,-36.903,30.045,-141.5109,0.5961,0.0000
C01138=-6.591,-39.512,31.092,-141.4605,0.4104,0.0000
C01139=-7.106,-42.459,31.903,-141.3865,0.2222,0.0000
C01140=-7.750,-45.198,32.306,-141.3268,-0.0353,0.0000
C01141=-9.416,-47.186,32.519,-141.4423,-0.9306,0.0000
C01142=-11.916,-48.107,32.693,-141.8310,-2.4259,0.0000
C01143=-14.756,-47.748,32.868,-142.5059,-4.1933,0.0000
C01144=-17.673,-46.769,32.984,-143.3894,-5.9463,0.0000
C01145=-20.574,-45.568,32.984,-156.5587,29.5172,0.0000
C01146=-23.329,-44.198,32.868,-154.4930,28.7476,0.0000
C01147=-25.591,-42.442,32.693,-152.6285,27.8084,0.0000
C01148=-26.708,-40.024,32.519,-151.2358,26.8826,0.0000
C01149=-26.480,-37.440,32.306,-150.5160,26.2498,0.0000
C01150=-24.998,-35.047,31.903,-150.3919,26.0100,0.0000
C01151=-23.279,-32.600,31.092,-150.3282,25.8161,0.0000
C01152=-21.772,-30.417,30.045,-150.2457,25.6386,0.0000
C01153=-20.769,-28.682,29.040,-150.1076,25.4525,0.0000
C01154=-20.608,-27.283,28.321,-149.8045,25.1396,0.0000
C01155=-21.662,-25.896,28.038,-149.2062,24.5133,0.0000
C01156=-22.835,-24.829,28.025,-149.2105,24.5706,0.0000
C01157=-23.852,-23.852,28.034,-150.5423,26.1858,0.0000
C01158=-24.829,-22.835,28.025,-151.9767,27.7448,0.0000
C01159=-25.896,-21.662,28.038,-152.0381,27.7619,0.0000
C01160=-27.283,-20.608,28.321,-151.5000,27.0845,0.0000
C01161=-28.682,-20.769,29.040,-151.2332,26.7435,0.0000
C01162=-30.417,-21.772,30.045,-151.0645,26.5778,0.0000
C01163=-32.600,-23.279,31.092,-150.8918,26.4630,0.0000
C01164=-35.047,-24.998,31.903,-150.6972,26.3606,0.0000
C01165=-37.440,-26.480,32.306,-150.4678,26.1944,0.0000
C01166=-40.024,-26.708,32.519,-149.9588,25.4168,0.0000
C01167=-42.442,-25.591,32.693,-149.2929,23.9951,0.0000
C01168=-44.198,-23.329,32.868,-148.7084,22.1817,0.0000
C01169=-45.568,-20.574,32.984,-148.3213,20.2537,0.0000
C01170=-46.769,-17.673,32.984,172.6068,36.3819,0.0000
C01171=-47.748,-14.756,32.868,174.7206,37.3765,0.0000
C01172=-48.107,-11.916,32.693,176.9157,38.1287,0.0000
C01173=-47.186,-9.416,32.519,178.8105,38.5518,0.0000
C01174=-45.198,-7.750,32.306,179.9553,38.6732,0.0000
C01175=-42.459,-7.106,31.903,-179.7150,38.6132,0.0000
C01176=-39.512,-6.591,31.092,-179.4747,38.5384,0.0000
C01177=-36.903,-6.113,30.045,-179.2379,38.4867,0.0000
C01178=-34.967,-5.595,29.040,-178.9526,38.4687,0.0000
C01179=-33.865,-4.720,28.321,-178.4219,38.4879,0.0000
C01180=-33.629,-2.994,28.038,-177.3634,38.5176,0.0000
C01181=-33.704,-1.410,28.025,-177.4234,38.5507,0.0000
C01182=-33.732,0.000,28.034,-179.9987,38.6152,0.0000
C01183=-33.704,1.410,28.025,177.4234,38.5508,0.0000
C01184=-33.629,2.994,28.038,177.3641,38.5176,0.0000
C01185=-33.865,4.720,28.321,178.4225,38.4879,0.0000
C01186=-34.967,5.595,29.040,178.9532,38.4687,0.0000
C01187=-36.903,6.113,30.045,179.2384,38.4866,0.0000
C01188=-39.512,6.591,31.092,179.4753,38.5384,0.0000
C01189=-42.459,7.106,31.903,179.7156,38.6131,0.0000
C01190=-45.198,7.750,32.306,-179.9547,38.6732,0.0000
C01191=-47.186,9.416,32.519,-178.8100,38.5517,0.0000
C01192=-48.107,11.916,32.693,-176.9155,38.1287,0.0000
C01193=-47.748,14.756,32.868,-174.7205,37.3765,0.0000
C01194=-46.769,17.673,32.984,-172.6067,36.3819,0.0000
C01195=-45.568,20.574,32.984,148.3213,20.2537,0.0000
C01196=-44.198,23.329,32.868,148.7085,22.1818,0.0000
C01197=-42.442,25.591,32.693,149.2930,23.9953,0.0000
C01198=-40.024,26.708,32.519,149.9590,25.4171,0.0000
C01199=-37.440,26.480,32.306,150.4681,26.1948,0.0000
C01200=-35.047,24.998,31.903,150.6974,26.3609,0.0000
C01201=-32.600,23.279,31.092,150.8921,26.4634,0.0000
C01202=-30.417,21.772,30.045,151.0648,26.5781,0.0000
C01203=-28.682,20.769,29.040,151.2334,26.7438,0.0000
C01204=-27.283,20.608,28.321,151.5004,27.0849,0.0000
C01205=-25.896,21.662,28.038,152.0385,27.7623,0.0000
C01206=-24.829,22.835,28.025,151.9767,27.7448,0.0000
C01207=-23.852,23.852,28.034,150.5437,26.1874,0.0000
C01208=-22.835,24.829,28.025,149.2105,24.5706,0.0000
C01209=-21.662,25.896,28.038,149.2066,24.5137,0.0000
C01210=-20.608,27.283,28.321,149.8048,25.1400,0.0000
C01211=-20.769,28.682,29.040,150.1079,25.4528,0.0000
C01212=-21.772,30.417,30.045,150.2461,25.6389,0.0000
C01213=-23.279,32.600,31.092,150.3285,25.8165,0.0000
C01214=-24.998,35.047,31.903,150.3922,26.0104,0.0000
C01215=-26.480,37.440,32.306,150.5163,26.2501,0.0000
C01216=-26.708,40.024,32.519,151.2361,26.8828,0.0000
C01217=-25.591,42.442,32.693,152.6287,27.8086,0.0000
C01218=-23.329,44.198,32.868,154.4930,28.7477,0.0000
C01219=-20.574,45.568,32.984,156.5587,29.5172,0.0000
C01220=-17.673,46.769,32.984,143.3894,-5.9463,0.0000
C01221=-14.756,47.748,32.868,142.5059,-4.1933,0.0000
C01222=-11.916,48.107,32.693,141.8310,-2.4259,0.0000
C01223=-9.416,47.186,32.519,141.4423,-0.9306,0.0000
C01224=-7.750,45.198,32.306,141.3268,-0.0353,0.0000
C01225=-7.106,42.459,31.903,141.3865,0.2222,0.0000
C01226=-6.591,39.512,31.092,141.4605,0.4104,0.0000
C01227=-6.113,36.903,30.045,141.5109,0.5961,0.0000
C01228=-5.595,34.967,29.040,141.5266,0.8196,0.0000
C01229=-4.720,33.865,28.321,141.5015,1.2347,0.0000
C01230=-2.994,33.629,28.038,141.4528,2.0621,0.0000
C01231=-1.410,33.704,28.025,141.4210,2.0148,0.0000
C01232=0.000,33.732,28.034,141.3848,-0.0010,0.0000
C01233=0.000,32.376,29.766,141.6284,-0.0012,0.0000
C01234=1.286,32.352,29.757,141.6633,-1.9630,0.0000
C01235=2.786,32.290,29.771,141.6939,-2.0532,0.0000
C01236=4.465,32.574,30.085,141.7380,-1.2416,0.0000
C01237=5.286,33.800,30.880,141.7545,-0.8533,0.0000
C01238=5.763,35.931,31.987,141.7241,-0.6525,0.0000
C01239=6.219,38.785,33.135,141.6499,-0.4820,0.0000
C01240=6.715,41.994,34.017,141.5427,-0.3079,0.0000
C01241=7.331,44.970,34.453,141.4446,-0.0687,0.0000
C01242=9.024,47.139,34.683,141.5316,0.8586,0.0000
C01243=11.608,48.163,34.870,141.9218,2.4394,0.0000
C01244=14.563,47.812,35.059,142.6423,4.3205,0.0000
C01245=17.608,46.795,35.183,143.6034,6.1807,0.0000
C01246=20.638,45.540,35.183,156.9199,-29.5556,0.0000
C01247=23.511,44.106,35.059,154.7051,-28.7583,0.0000
C01248=25.848,42.264,34.870,152.7180,-27.7620,0.0000
C01249=26.951,39.714,34.683,151.2646,-26.7709,0.0000
C01250=26.615,36.982,34.453,150.5483,-26.0957,0.0000
C01251=24.946,34.442,34.017,150.4705,-25.8468,0.0000
C01252=23.028,31.823,33.135,150.4455,-25.6435,0.0000
C01253=21.332,29.482,31.987,150.3941,-25.4634,0.0000
C01254=20.163,27.638,30.880,150.2841,-25.2864,0.0000
C01255=19.876,26.191,30.085,150.0066,-24.9899,0.0000
C01256=20.863,24.802,29.771,149.4226,-24.3741,0.0000
C01257=21.967,23.786,29.757,149.4563,-24.4643,0.0000
C01258=22.894,22.894,29.766,150.7557,-26.0355,0.0000
C01259=23.786,21.968,29.757,152.1535,-27.5531,0.0000
C01260=24.802,20.862,29.771,152.2437,-27.6038,0.0000
C01261=26.191,19.876,30.085,151.7123,-26.9424,0.0000
C01262=27.638,20.163,30.880,151.4563,-26.6281,0.0000
C01263=29.482,21.332,31.987,151.2903,-26.4896,0.0000
C01264=31.823,23.028,33.135,151.1073,-26.4017,0.0000
C01265=34.442,24.946,34.017,150.8930,-26.3312,0.0000
C01266=36.982,26.615,34.453,150.6423,-26.2035,0.0000
C01267=39.714,26.951,34.683,150.0856,-25.4186,0.0000
C01268=42.264,25.848,34.870,149.3627,-23.9290,0.0000
C01269=44.106,23.511,35.059,148.7420,-21.9980,0.0000
C01270=45.540,20.638,35.183,148.3506,-19.9382,0.0000
C01271=46.795,17.608,35.183,-172.3375,-36.1515,0.0000
C01272=47.812,14.563,35.059,-174.5705,-37.2335,0.0000
C01273=48.163,11.608,34.870,-176.9022,-38.0375,0.0000
C01274=47.139,9.024,34.683,-178.9035,-38.4633,0.0000
C01275=44.970,7.331,34.453,179.9122,-38.5554,0.0000
C01276=41.994,6.715,34.017,179.6068,-38.4567,0.0000
C01277=38.785,6.219,33.135,179.3854,-38.3485,0.0000
C01278=35.931,5.763,31.987,179.1688,-38.2730,0.0000
C01279=33.800,5.286,30.880,178.9135,-38.2405,0.0000
C01280=32.574,4.465,30.085,178.4189,-38.2514,0.0000
C01281=32.290,2.786,29.771,177.3842,-38.2770,0.0000
C01282=32.352,1.286,29.757,177.4980,-38.3101,0.0000
C01283=32.376,0.000,29.766,179.9984,-38.3716,0.0000
C01284=32.352,-1.286,29.757,-177.4979,-38.3101,0.0000
C01285=32.290,-2.786,29.771,-177.3849,-38.2770,0.0000
C01286=32.574,-4.465,30.085,-178.4195,-38.2514,0.0000
C01287=33.800,-5.286,30.880,-178.9141,-38.2405,0.0000
C01288=35.931,-5.763,31.987,-179.1693,-38.2729,0.0000
C01289=38.785,-6.219,33.135,-179.3859,-38.3485,0.0000
C01290=41.994,-6.715,34.017,-179.6074,-38.4566,0.0000
C01291=44.970,-7.331,34.453,-179.9127,-38.5553,0.0000
C01292=47.139,-9.024,34.683,178.9030,-38.4632,0.0000
C01293=48.163,-11.608,34.870,176.9020,-38.0375,0.0000
C01294=47.812,-14.563,35.059,174.5704,-37.2335,0.0000
C01295=46.795,-17.608,35.183,172.3375,-36.1515,0.0000
C01296=45.540,-20.638,35.183,-148.3506,-19.9383,0.0000
C01297=44.106,-23.511,35.059,-148.7420,-21.9981,0.0000
C01298=42.264,-25.848,34.870,-149.3628,-23.9292,0.0000
C01299=39.714,-26.951,34.683,-150.0858,-25.4190,0.0000
C01300=36.982,-26.615,34.453,-150.6426,-26.2039,0.0000
C01301=34.442,-24.946,34.017,-150.8933,-26.3316,0.0000
C01302=31.823,-23.028,33.135,-151.1075,-26.4021,0.0000
C01303=29.482,-21.332,31.987,-151.2906,-26.4900,0.0000
C01304=27.638,-20.163,30.880,-151.4566,-26.6285,0.0000
C01305=26.191,-19.876,30.085,-151.7126,-26.9428,0.0000
C01306=24.802,-20.863,29.771,-152.2442,-27.6042,0.0000
C01307=23.786,-21.967,29.757,-152.1535,-27.5530,0.0000
C01308=22.894,-22.894,29.766,-150.7574,-26.0374,0.0000
C01309=21.968,-23.786,29.757,-149.4563,-24.4643,0.0000
C01310=20.862,-24.802,29.771,-149.4230,-24.3746,0.0000
C01311=19.876,-26.191,30.085,-150.0069,-24.9902,0.0000
C01312=20.163,-27.638,30.880,-150.2844,-25.2867,0.0000
C01313=21.332,-29.482,31.987,-150.3944,-25.4637,0.0000
C01314=23.028,-31.823,33.135,-150.4458,-25.6438,0.0000
C01315=24.946,-34.442,34.017,-150.4709,-25.8471,0.0000
C01316=26.615,-36.982,34.453,-150.5487,-26.0960,0.0000
C01317=26.951,-39.714,34.683,-151.2649,-26.7712,0.0000
C01318=25.848,-42.264,34.870,-152.7182,-27.7621,0.0000
C01319=23.511,-44.106,35.059,-154.7052,-28.7583,0.0000
C01320=20.638,-45.540,35.183,-156.9199,-29.5556,0.0000
C01321=17.608,-46.795,35.183,-143.6034,6.1807,0.0000
C01322=14.563,-47.812,35.059,-142.6423,4.3205,0.0000
C01323=11.608,-48.163,34.870,-141.9218,2.4394,0.0000
C01324=9.024,-47.139,34.683,-141.5316,0.8586,0.0000
C01325=7.331,-44.970,34.453,-141.4446,-0.0687,0.0000
C01326=6.715,-41.994,34.017,-141.5427,-0.3079,0.0000
C01327=6.219,-38.785,33.135,-141.6499,-0.4820,0.0000
C01328=5.763,-35.931,31.987,-141.7241,-0.6525,0.0000
C01329=5.286,-33.800,30.880,-141.7545,-0.8533,0.0000
C01330=4.465,-32.574,30.085,-141.7380,-1.2416,0.0000
C01331=2.786,-32.290,29.771,-141.6939,-2.0532,0.0000
C01332=1.286,-32.352,29.757,-141.6633,-1.9630,0.0000
C01333=0.000,-32.376,29.766,-141.6284,-0.0012,0.0000
C01334=0.000,-32.376,29.766,-141.6284,-0.0012,0.0000
C01335=-1.286,-32.352,29.757,-141.6633,1.9630,0.0000
C01336=-2.786,-32.290,29.771,-141.6939,2.0526,0.0000
C01337=-4.465,-32.574,30.085,-141.7380,1.2411,0.0000
C01338=-5.286,-33.800,30.880,-141.7545,0.8529,0.0000
C01339=-5.763,-35.931,31.987,-141.7241,0.6521,0.0000
C01340=-6.219,-38.785,33.135,-141.6499,0.4816,0.0000
C01341=-6.715,-41.994,34.017,-141.5427,0.3074,0.0000
C01342=-7.331,-44.970,34.453,-141.4446,0.0682,0.0000
C01343=-9.024,-47.139,34.683,-141.5317,-0.8589,0.0000
C01344=-11.608,-48.163,34.870,-141.9219,-2.4396,0.0000
C01345=-14.563,-47.812,35.059,-142.6423,-4.3206,0.0000
C01346=-17.608,-46.795,35.183,-143.6034,-6.1807,0.0000
C01347=-20.638,-45.540,35.183,-156.9199,29.5556,0.0000
C01348=-23.511,-44.106,35.059,-154.7051,28.7583,0.0000
C01349=-25.848,-42.264,34.870,-152.7180,27.7620,0.0000
C01350=-26.951,-39.714,34.683,-151.2646,26.7709,0.0000
C01351=-26.615,-36.982,34.453,-150.5483,26.0957,0.0000
C01352=-24.946,-34.442,34.017,-150.4705,25.8468,0.0000
C01353=-23.028,-31.823,33.135,-150.4455,25.6435,0.0000
C01354=-21.332,-29.482,31.987,-150.3941,25.4634,0.0000
C01355=-20.163,-27.638,30.880,-150.2841,25.2864,0.0000
C01356=-19.876,-26.191,30.085,-150.0066,24.9899,0.0000
C01357=-20.863,-24.802,29.771,-149.4226,24.3741,0.0000
C01358=-21.967,-23.786,29.757,-149.4563,24.4643,0.0000
C01359=-22.894,-22.894,29.766,-150.7557,26.0355,0.0000
C01360=-23.786,-21.968,29.757,-152.1535,27.5531,0.0000
C01361=-24.802,-20.862,29.771,-152.2437,27.6038,0.0000
C01362=-26.191,-19.876,30.085,-151.7123,26.9424,0.0000
C01363=-27.638,-20.163,30.880,-151.4563,26.6281,0.0000
C01364=-29.482,-21.332,31.987,-151.2903,26.4896,0.0000
C01365=-31.823,-23.028,33.135,-151.1073,26.4017,0.0000
C01366=-34.442,-24.946,34.017,-150.8930,26.3312,0.0000
C01367=-36.982,-26.615,34.453,-150.6423,26.2035,0.0000
C01368=-39.714,-26.951,34.683,-150.0856,25.4186,0.0000
C01369=-42.264,-25.848,34.870,-149.3627,23.9290,0.0000
C01370=-44.106,-23.511,35.059,-148.7420,21.9980,0.0000
C01371=-45.540,-20.638,35.183,-148.3506,19.9382,0.0000
C01372=-46.795,-17.608,35.183,172.3375,36.1515,0.0000
C01373=-47.812,-14.563,35.059,174.5705,37.2335,0.0000
C01374=-48.163,-11.608,34.870,176.9022,38.0375,0.0000
C01375=-47.139,-9.024,34.683,178.9035,38.4633,0.0000
C01376=-44.970,-7.331,34.453,-179.9122,38.5554,0.0000
C01377=-41.994,-6.715,34.017,-179.6068,38.4567,0.0000
C01378=-38.785,-6.219,33.135,-179.3854,38.3485,0.0000
C01379=-35.931,-5.763,31.987,-179.1688,38.2730,0.0000
C01380=-33.800,-5.286,30.880,-178.9135,38.2405,0.0000
C01381=-32.574,-4.465,30.085,-178.4189,38.2514,0.0000
C01382=-32.290,-2.786,29.771,-177.3842,38.2770,0.0000
C01383=-32.352,-1.286,29.757,-177.4980,38.3101,0.0000
C01384=-32.376,0.000,29.766,-179.9984,38.3716,0.0000
C01385=-32.352,1.286,29.757,177.4979,38.3101,0.0000
C01386=-32.290,2.786,29.771,177.3849,38.2770,0.0000
C01387=-32.574,4.465,30.085,178.4195,38.2514,0.0000
C01388=-33.800,5.286,30.880,178.9141,38.2405,0.0000
C01389=-35.931,5.763,31.987,179.1693,38.2729,0.0000
C01390=-38.785,6.219,33.135,179.3859,38.3485,0.0000
C01391=-41.994,6.715,34.017,179.6074,38.4566,0.0000
C01392=-44.970,7.331,34.453,179.9127,38.5553,0.0000
C01393=-47.139,9.024,34.683,-178.9030,38.4632,0.0000
C01394=-48.163,11.608,34.870,-176.9020,38.0375,0.0000
C01395=-47.812,14.563,35.059,-174.5704,37.2335,0.0000
C01396=-46.795,17.608,35.183,-172.3375,36.1515,0.0000
C01397=-45.540,20.638,35.183,148.3506,19.9383,0.0000
C01398=-44.106,23.511,35.059,148.7420,21.9981,0.0000
C01399=-42.264,25.848,34.870,149.3628,23.9292,0.0000
C01400=-39.714,26.951,34.683,150.0858,25.4190,0.0000
C01401=-36.982,26.615,34.453,150.6426,26.2039,0.0000
C01402=-34.442,24.946,34.017,150.8933,26.3316,0.0000
C01403=-31.823,23.028,33.135,151.1075,26.4021,0.0000
C01404=-29.482,21.332,31.987,151.2906,26.4900,0.0000
C01405=-27.638,20.163,30.880,151.4566,26.6285,0.0000
C01406=-26.191,19.876,30.085,151.7126,26.9428,0.0000
C01407=-24.802,20.863,29.771,152.2442,27.6042,0.0000
C01408=-23.786,21.967,29.757,152.1535,27.5530,0.0000
C01409=-22.894,22.894,29.766,150.7574,26.0374,0.0000
C01410=-21.968,23.786,29.757,149.4563,24.4643,0.0000
C01411=-20.862,24.802,29.771,149.4230,24.3746,0.0000
C01412=-19.876,26.191,30.085,150.0069,24.9902,0.0000
C01413=-20.163,27.638,30.880,150.2844,25.2867,0.0000
C01414=-21.332,29.482,31.987,150.3944,25.4637,0.0000
C01415=-23.028,31.823,33.135,150.4458,25.6438,0.0000
C01416=-24.946,34.442,34.017,150.4709,25.8471,0.0000
C01417=-26.615,36.982,34.453,150.5487,26.0960,0.0000
C01418=-26.951,39.714,34.683,151.2649,26.7712,0.0000
C01419=-25.848,42.264,34.870,152.7182,27.7621,0.0000
C01420=-23.511,44.106,35.059,154.7052,28.7583,0.0000
C01421=-20.638,45.540,35.183,156.9199,29.5556,0.0000
C01422=-17.608,46.795,35.183,143.6034,-6.1807,0.0000
C01423=-14.563,47.812,35.059,142.6423,-4.3206,0.0000
C01424=-11.608,48.163,34.870,141.9219,-2.4396,0.0000
C01425=-9.024,47.139,34.683,141.5317,-0.8589,0.0000
C01426=-7.331,44.970,34.453,141.4446,0.0682,0.0000
C01427=-6.715,41.994,34.017,141.5427,0.3074,0.0000
C01428=-6.219,38.785,33.135,141.6499,0.4816,0.0000
C01429=-5.763,35.931,31.987,141.7241,0.6521,0.0000
C01430=-5.286,33.800,30.880,141.7545,0.8529,0.0000
C01431=-4.465,32.574,30.085,141.7380,1.2411,0.0000
C01432=-2.786,32.290,29.771,141.6939,2.0526,0.0000
C01433=-1.286,32.352,29.757,141.6633,1.9630,0.0000
C01434=0.000,32.376,29.766,141.6284,-0.0012,0.0000
C01435=0.000,31.053,31.524,141.9059,-0.0015,0.0000
C01436=1.165,31.033,31.514,141.9394,-1.9071,0.0000
C01437=2.582,30.983,31.529,141.9691,-2.0439,0.0000
C01438=4.218,31.318,31.874,142.0087,-1.2492,0.0000
C01439=4.987,32.673,32.745,142.0169,-0.8870,0.0000
C01440=5.430,35.005,33.954,141.9715,-0.7068,0.0000
C01441=5.871,38.106,35.198,141.8726,-0.5483,0.0000
C01442=6.356,41.567,36.145,141.7309,-0.3846,0.0000
C01443=6.949,44.762,36.610,141.5936,-0.1605,0.0000
C01444=8.669,47.097,36.854,141.6515,0.8007,0.0000
C01445=11.329,48.213,37.052,142.0431,2.4664,0.0000
C01446=14.389,47.870,37.251,142.8105,4.4576,0.0000
C01447=17.550,46.817,37.382,143.8507,6.4178,0.0000
C01448=20.695,45.514,37.382,157.3120,-29.5736,0.0000
C01449=23.675,44.023,37.251,154.9522,-28.7558,0.0000
C01450=26.081,42.103,37.052,152.8437,-27.7067,0.0000
C01451=27.172,39.432,36.854,151.3297,-26.6512,0.0000
C01452=26.738,36.565,36.610,150.6160,-25.9316,0.0000
C01453=24.898,33.886,36.145,150.5829,-25.6705,0.0000
C01454=22.793,31.096,35.198,150.5948,-25.4542,0.0000
C01455=20.912,28.592,33.954,150.5730,-25.2684,0.0000
C01456=19.577,26.630,32.745,150.4899,-25.0985,0.0000
C01457=19.163,25.127,31.874,150.2372,-24.8178,0.0000
C01458=20.082,23.734,31.529,149.6679,-24.2137,0.0000
C01459=21.120,22.768,31.514,149.7339,-24.3402,0.0000
C01460=21.958,21.958,31.524,150.9983,-25.8639,0.0000
C01461=22.768,21.120,31.514,152.3567,-27.3368,0.0000
C01462=23.734,20.082,31.529,152.4788,-27.4241,0.0000
C01463=25.127,19.163,31.874,151.9548,-26.7796,0.0000
C01464=26.630,19.577,32.745,151.7094,-26.4913,0.0000
C01465=28.592,20.912,33.954,151.5445,-26.3785,0.0000
C01466=31.096,22.793,35.198,151.3481,-26.3157,0.0000
C01467=33.886,24.898,36.145,151.1109,-26.2750,0.0000
C01468=36.565,26.738,36.610,150.8362,-26.1838,0.0000
C01469=39.432,27.172,36.854,150.2297,-25.3908,0.0000
C01470=42.103,26.081,37.052,149.4498,-23.8337,0.0000
C01471=44.023,23.675,37.251,148.7961,-21.7872,0.0000
C01472=45.514,20.695,37.382,148.4058,-19.6007,0.0000
C01473=46.817,17.550,37.382,-172.0698,-35.8874,0.0000
C01474=47.870,14.389,37.251,-174.4110,-37.0581,0.0000
C01475=48.213,11.329,37.052,-176.8731,-37.9155,0.0000
C01476=47.097,8.669,36.854,-178.9791,-38.3441,0.0000
C01477=44.762,6.949,36.610,179.7952,-38.4062,0.0000
C01478=41.567,6.356,36.145,179.5102,-38.2681,0.0000
C01479=38.106,5.871,35.198,179.3031,-38.1253,0.0000
C01480=35.005,5.430,33.954,179.1028,-38.0250,0.0000
C01481=32.673,4.987,32.745,178.8747,-37.9777,0.0000
C01482=31.318,4.218,31.874,178.4151,-37.9806,0.0000
C01483=30.983,2.582,31.529,177.4058,-38.0024,0.0000
C01484=31.033,1.165,31.514,177.5784,-38.0357,0.0000
C01485=31.053,0.000,31.524,179.9982,-38.0941,0.0000
C01486=31.033,-1.165,31.514,-177.5781,-38.0358,0.0000
C01487=30.983,-2.582,31.529,-177.4066,-38.0024,0.0000
C01488=31.318,-4.218,31.874,-178.4157,-37.9806,0.0000
C01489=32.673,-4.987,32.745,-178.8753,-37.9777,0.0000
C01490=35.005,-5.430,33.954,-179.1033,-38.0250,0.0000
C01491=38.106,-5.871,35.198,-179.3036,-38.1253,0.0000
C01492=41.567,-6.356,36.145,-179.5108,-38.2680,0.0000
C01493=44.762,-6.949,36.610,-179.7958,-38.4062,0.0000
C01494=47.097,-8.669,36.854,178.9786,-38.3440,0.0000
C01495=48.213,-11.329,37.052,176.8728,-37.9154,0.0000
C01496=47.870,-14.389,37.251,174.4109,-37.0581,0.0000
C01497=46.817,-17.550,37.382,172.0697,-35.8874,0.0000
C01498=45.514,-20.695,37.382,-148.4059,-19.6007,0.0000
C01499=44.023,-23.675,37.251,-148.7961,-21.7873,0.0000
C01500=42.103,-26.081,37.052,-149.4499,-23.8339,0.0000
C01501=39.432,-27.172,36.854,-150.2299,-25.3911,0.0000
C01502=36.565,-26.738,36.610,-150.8364,-26.1842,0.0000
C01503=33.886,-24.898,36.145,-151.1112,-26.2754,0.0000
C01504=31.096,-22.793,35.198,-151.3484,-26.3160,0.0000
C01505=28.592,-20.912,33.954,-151.5448,-26.3788,0.0000
C01506=26.630,-19.577,32.745,-151.7097,-26.4917,0.0000
C01507=25.127,-19.163,31.874,-151.9551,-26.7800,0.0000
C01508=23.734,-20.082,31.529,-152.4792,-27.4246,0.0000
C01509=22.768,-21.120,31.514,-152.3565,-27.3366,0.0000
C01510=21.958,-21.958,31.524,-151.0003,-25.8662,0.0000
C01511=21.120,-22.768,31.514,-149.7337,-24.3401,0.0000
C01512=20.082,-23.734,31.529,-149.6683,-24.2142,0.0000
C01513=19.163,-25.127,31.874,-150.2376,-24.8182,0.0000
C01514=19.577,-26.630,32.745,-150.4902,-25.0988,0.0000
C01515=20.912,-28.592,33.954,-150.5733,-25.2688,0.0000
C01516=22.793,-31.096,35.198,-150.5952,-25.4546,0.0000
C01517=24.898,-33.886,36.145,-150.5832,-25.6708,0.0000
C01518=26.738,-36.565,36.610,-150.6164,-25.9319,0.0000
C01519=27.172,-39.432,36.854,-151.3300,-26.6515,0.0000
C01520=26.081,-42.103,37.052,-152.8439,-27.7068,0.0000
C01521=23.675,-44.023,37.251,-154.9523,-28.7558,0.0000
C01522=20.695,-45.514,37.382,-157.3120,-29.5736,0.0000
C01523=17.550,-46.817,37.382,-143.8507,6.4178,0.0000
C01524=14.389,-47.870,37.251,-142.8105,4.4576,0.0000
C01525=11.329,-48.213,37.052,-142.0431,2.4664,0.0000
C01526=8.669,-47.097,36.854,-141.6515,0.8007,0.0000
C01527=6.949,-44.762,36.610,-141.5936,-0.1605,0.0000
C01528=6.356,-41.567,36.145,-141.7309,-0.3846,0.0000
C01529=5.871,-38.106,35.198,-141.8726,-0.5483,0.0000
C01530=5.430,-35.005,33.954,-141.9715,-0.7068,0.0000
C01531=4.987,-32.673,32.745,-142.0169,-0.8870,0.0000
C01532=4.218,-31.318,31.874,-142.0087,-1.2492,0.0000
C01533=2.582,-30.983,31.529,-141.9691,-2.0439,0.0000
C01534=1.165,-31.033,31.514,-141.9394,-1.9071,0.0000
C01535=0.000,-31.053,31.524,-141.9059,-0.0015,0.0000
C01536=0.000,-31.053,31.524,-141.9059,-0.0015,0.0000
C01537=-1.165,-31.033,31.514,-141.9394,1.9073,0.0000
C01538=-2.582,-30.983,31.529,-141.9691,2.0433,0.0000
C01539=-4.218,-31.318,31.874,-142.0088,1.2487,0.0000
C01540=-4.987,-32.673,32.745,-142.0169,0.8865,0.0000
C01541=-5.430,-35.005,33.954,-141.9716,0.7063,0.0000
C01542=-5.871,-38.106,35.198,-141.8727,0.5478,0.0000
C01543=-6.356,-41.567,36.145,-141.7309,0.3841,0.0000
C01544=-6.949,-44.762,36.610,-141.5936,0.1600,0.0000
C01545=-8.669,-47.097,36.854,-141.6516,-0.8011,0.0000
C01546=-11.329,-48.213,37.052,-142.0432,-2.4666,0.0000
C01547=-14.389,-47.870,37.251,-142.8105,-4.4577,0.0000
C01548=-17.550,-46.817,37.382,-143.8507,-6.4178,0.0000
C01549=-20.695,-45.514,37.382,-157.3120,29.5736,0.0000
C01550=-23.675,-44.023,37.251,-154.9522,28.7558,0.0000
C01551=-26.081,-42.103,37.052,-152.8437,27.7067,0.0000
C01552=-27.172,-39.432,36.854,-151.3297,26.6512,0.0000
C01553=-26.738,-36.565,36.610,-150.6160,25.9316,0.0000
C01554=-24.898,-33.886,36.145,-150.5829,25.6705,0.0000
C01555=-22.793,-31.096,35.198,-150.5948,25.4542,0.0000
C01556=-20.912,-28.592,33.954,-150.5730,25.2684,0.0000
C01557=-19.577,-26.630,32.745,-150.4899,25.0985,0.0000
C01558=-19.163,-25.127,31.874,-150.2372,24.8178,0.0000
C01559=-20.082,-23.734,31.529,-149.6679,24.2137,0.0000
C01560=-21.120,-22.768,31.514,-149.7339,24.3402,0.0000
C01561=-21.958,-21.958,31.524,-150.9983,25.8639,0.0000
C01562=-22.768,-21.120,31.514,-152.3567,27.3368,0.0000
C01563=-23.734,-20.082,31.529,-152.4788,27.4241,0.0000
C01564=-25.127,-19.163,31.874,-151.9548,26.7796,0.0000
C01565=-26.630,-19.577,32.745,-151.7094,26.4913,0.0000
C01566=-28.592,-20.912,33.954,-151.5445,26.3785,0.0000
C01567=-31.096,-22.793,35.198,-151.3481,26.3157,0.0000
C01568=-33.886,-24.898,36.145,-151.1109,26.2750,0.0000
C01569=-36.565,-26.738,36.610,-150.8362,26.1838,0.0000
C01570=-39.432,-27.172,36.854,-150.2297,25.3908,0.0000
C01571=-42.103,-26.081,37.052,-149.4498,23.8337,0.0000
C01572=-44.023,-23.675,37.251,-148.7961,21.7872,0.0000
C01573=-45.514,-20.695,37.382,-148.4058,19.6007,0.0000
C01574=-46.817,-17.550,37.382,172.0698,35.8874,0.0000
C01575=-47.870,-14.389,37.251,174.4110,37.0581,0.0000
C01576=-48.213,-11.329,37.052,176.8731,37.9155,0.0000
C01577=-47.097,-8.669,36.854,178.9791,38.3441,0.0000
C01578=-44.762,-6.949,36.610,-179.7952,38.4062,0.0000
C01579=-41.567,-6.356,36.145,-179.5102,38.2681,0.0000
C01580=-38.106,-5.871,35.198,-179.3031,38.1253,0.0000
C01581=-35.005,-5.430,33.954,-179.1028,38.0250,0.0000
C01582=-32.673,-4.987,32.745,-178.8747,37.9777,0.0000
C01583=-31.318,-4.218,31.874,-178.4151,37.9806,0.0000
C01584=-30.983,-2.582,31.529,-177.4058,38.0024,0.0000
C01585=-31.033,-1.165,31.514,-177.5784,38.0357,0.0000
C01586=-31.053,0.000,31.524,-179.9982,38.0941,0.0000
C01587=-31.033,1.165,31.514,177.5781,38.0358,0.0000
C01588=-30.983,2.582,31.529,177.4066,38.0024,0.0000
C01589=-31.318,4.218,31.874,178.4157,37.9806,0.0000
C01590=-32.673,4.987,32.745,178.8753,37.9777,0.0000
C01591=-35.005,5.430,33.954,179.1033,38.0250,0.0000
C01592=-38.106,5.871,35.198,179.3036,38.1253,0.0000
C01593=-41.567,6.356,36.145,179.5108,38.2680,0.0000
C01594=-44.762,6.949,36.610,179.7958,38.4062,0.0000
C01595=-47.097,8.669,36.854,-178.9786,38.3440,0.0000
C01596=-48.213,11.329,37.052,-176.8728,37.9154,0.0000
C01597=-47.870,14.389,37.251,-174.4109,37.0581,0.0000
C01598=-46.817,17.550,37.382,-172.0697,35.8874,0.0000
C01599=-45.514,20.695,37.382,148.4059,19.6007,0.0000
C01600=-44.023,23.675,37.251,148.7961,21.7873,0.0000
C01601=-42.103,26.081,37.052,149.4499,23.8339,0.0000
C01602=-39.432,27.172,36.854,150.2299,25.3911,0.0000
C01603=-36.565,26.738,36.610,150.8364,26.1842,0.0000
C01604=-33.886,24.898,36.145,151.1112,26.2754,0.0000
C01605=-31.096,22.793,35.198,151.3484,26.3160,0.0000
C01606=-28.592,20.912,33.954,151.5448,26.3788,0.0000
C01607=-26.630,19.577,32.745,151.7097,26.4917,0.0000
C01608=-25.127,19.163,31.874,151.9551,26.7800,0.0000
C01609=-23.734,20.082,31.529,152.4792,27.4246,0.0000
C01610=-22.768,21.120,31.514,152.3565,27.3366,0.0000
C01611=-21.958,21.958,31.524,151.0003,25.8662,0.0000
C01612=-21.120,22.768,31.514,149.7337,24.3401,0.0000
C01613=-20.082,23.734,31.529,149.6683,24.2142,0.0000
C01614=-19.163,25.127,31.874,150.2376,24.8182,0.0000
C01615=-19.577,26.630,32.745,150.4902,25.0988,0.0000
C01616=-20.912,28.592,33.954,150.5733,25.2688,0.0000
C01617=-22.793,31.096,35.198,150.5952,25.4546,0.0000
C01618=-24.898,33.886,36.145,150.5832,25.6708,0.0000
C01619=-26.738,36.565,36.610,150.6164,25.9319,0.0000
C01620=-27.172,39.432,36.854,151.3300,26.6515,0.0000
C01621=-26.081,42.103,37.052,152.8439,27.7068,0.0000
C01622=-23.675,44.023,37.251,154.9523,28.7558,0.0000
C01623=-20.695,45.514,37.382,157.3120,29.5736,0.0000
C01624=-17.550,46.817,37.382,143.8507,-6.4178,0.0000
C01625=-14.389,47.870,37.251,142.8105,-4.4577,0.0000
C01626=-11.329,48.213,37.052,142.0432,-2.4666,0.0000
C01627=-8.669,47.097,36.854,141.6516,-0.8011,0.0000
C01628=-6.949,44.762,36.610,141.5936,0.1600,0.0000
C01629=-6.356,41.567,36.145,141.7309,0.3841,0.0000
C01630=-5.871,38.106,35.198,141.8727,0.5478,0.0000
C01631=-5.430,35.005,33.954,141.9716,0.7063,0.0000
C01632=-4.987,32.673,32.745,142.0169,0.8865,0.0000
C01633=-4.218,31.318,31.874,142.0088,1.2487,0.0000
C01634=-2.582,30.983,31.529,141.9691,2.0433,0.0000
C01635=-1.165,31.033,31.514,141.9394,1.9073,0.0000
C01636=0.000,31.053,31.524,141.9059,-0.0015,0.0000
C01637=0.000,29.775,33.314,142.2164,-0.0017,0.0000
C01638=1.048,29.759,33.303,142.2483,-1.8474,0.0000
C01639=2.386,29.720,33.319,142.2773,-2.0340,0.0000
C01640=3.979,30.109,33.696,142.3127,-1.2565,0.0000
C01641=4.702,31.601,34.645,142.3126,-0.9188,0.0000
C01642=5.119,34.140,35.953,142.2518,-0.7560,0.0000
C01643=5.555,37.486,37.285,142.1271,-0.6052,0.0000
C01644=6.036,41.186,38.288,141.9501,-0.4472,0.0000
C01645=6.613,44.579,38.776,141.7735,-0.2340,0.0000
C01646=8.359,47.059,39.032,141.8025,0.7627,0.0000
C01647=11.087,48.257,39.238,142.1966,2.5124,0.0000
C01648=14.238,47.919,39.446,143.0124,4.6080,0.0000
C01649=17.499,46.837,39.582,144.1323,6.6582,0.0000
C01650=20.745,45.492,39.582,157.7361,-29.5707,0.0000
C01651=23.816,43.952,39.446,155.2383,-28.7414,0.0000
C01652=26.283,41.963,39.238,153.0108,-27.6458,0.0000
C01653=27.365,39.186,39.032,151.4357,-26.5277,0.0000
C01654=26.846,36.198,38.776,150.7231,-25.7628,0.0000
C01655=24.854,33.391,38.288,150.7313,-25.4860,0.0000
C01656=22.579,30.435,37.285,150.7776,-25.2525,0.0000
C01657=20.521,27.760,35.953,150.7832,-25.0569,0.0000
C01658=19.020,25.670,34.645,150.7252,-24.8912,0.0000
C01659=18.476,24.104,33.696,150.4961,-24.6252,0.0000
C01660=19.328,22.702,33.319,149.9416,-24.0332,0.0000
C01661=20.302,21.784,33.303,150.0418,-24.1985,0.0000
C01662=21.054,21.054,33.314,151.2689,-25.6714,0.0000
C01663=21.784,20.302,33.303,152.5850,-27.0967,0.0000
C01664=22.702,19.328,33.320,152.7415,-27.2229,0.0000
C01665=24.104,18.476,33.696,152.2255,-26.5953,0.0000
C01666=25.670,19.020,34.645,151.9896,-26.3319,0.0000
C01667=27.760,20.521,35.953,151.8233,-26.2426,0.0000
C01668=30.435,22.579,37.285,151.6099,-26.2022,0.0000
C01669=33.391,24.854,38.288,151.3459,-26.1884,0.0000
C01670=36.198,26.846,38.776,151.0443,-26.1304,0.0000
C01671=39.186,27.365,39.032,150.3874,-25.3280,0.0000
C01672=41.963,26.283,39.238,149.5519,-23.7038,0.0000
C01673=43.952,23.816,39.446,148.8699,-21.5457,0.0000
C01674=45.492,20.745,39.582,148.4870,-19.2399,0.0000
C01675=46.837,17.499,39.582,-171.8030,-35.5888,0.0000
C01676=47.919,14.238,39.446,-174.2382,-36.8483,0.0000
C01677=48.257,11.087,39.238,-176.8215,-37.7607,0.0000
C01678=47.059,8.359,39.032,-179.0296,-38.1935,0.0000
C01679=44.579,6.613,38.776,179.7021,-38.2262,0.0000
C01680=41.186,6.036,38.288,179.4321,-38.0486,0.0000
C01681=37.486,5.555,37.285,179.2333,-37.8704,0.0000
C01682=34.140,5.119,35.953,179.0439,-37.7444,0.0000
C01683=31.601,4.702,34.645,178.8390,-37.6817,0.0000
C01684=30.109,3.979,33.696,178.4123,-37.6766,0.0000
C01685=29.720,2.386,33.319,177.4291,-37.6947,0.0000
C01686=29.759,1.048,33.303,177.6640,-37.7286,0.0000
C01687=29.775,0.000,33.314,179.9979,-37.7836,0.0000
C01688=29.759,-1.048,33.303,-177.6635,-37.7286,0.0000
C01689=29.720,-2.386,33.320,-177.4299,-37.6948,0.0000
C01690=30.109,-3.979,33.696,-178.4130,-37.6766,0.0000
C01691=31.601,-4.702,34.645,-178.8395,-37.6817,0.0000
C01692=34.140,-5.119,35.953,-179.0444,-37.7443,0.0000
C01693=37.486,-5.555,37.285,-179.2338,-37.8704,0.0000
C01694=41.186,-6.036,38.288,-179.4326,-38.0485,0.0000
C01695=44.579,-6.613,38.776,-179.7027,-38.2261,0.0000
C01696=47.059,-8.359,39.032,179.0291,-38.1934,0.0000
C01697=48.257,-11.087,39.238,176.8212,-37.7607,0.0000
C01698=47.919,-14.238,39.446,174.2381,-36.8483,0.0000
C01699=46.837,-17.499,39.582,171.8030,-35.5888,0.0000
C01700=45.492,-20.745,39.582,-148.4871,-19.2399,0.0000
C01701=43.952,-23.816,39.446,-148.8700,-21.5457,0.0000
C01702=41.963,-26.283,39.238,-149.5520,-23.7040,0.0000
C01703=39.186,-27.365,39.032,-150.3876,-25.3284,0.0000
C01704=36.198,-26.846,38.776,-151.0446,-26.1308,0.0000
C01705=33.391,-24.854,38.288,-151.3462,-26.1888,0.0000
C01706=30.435,-22.579,37.285,-151.6102,-26.2026,0.0000
C01707=27.760,-20.521,35.953,-151.8236,-26.2429,0.0000
C01708=25.670,-19.020,34.645,-151.9899,-26.3322,0.0000
C01709=24.104,-18.476,33.696,-152.2258,-26.5957,0.0000
C01710=22.702,-19.328,33.319,-152.7420,-27.2234,0.0000
C01711=21.784,-20.302,33.303,-152.5848,-27.0964,0.0000
C01712=21.054,-21.054,33.314,-151.2712,-25.6741,0.0000
C01713=20.302,-21.784,33.303,-150.0415,-24.1982,0.0000
C01714=19.328,-22.702,33.320,-149.9420,-24.0337,0.0000
C01715=18.476,-24.104,33.696,-150.4965,-24.6256,0.0000
C01716=19.020,-25.670,34.645,-150.7255,-24.8916,0.0000
C01717=20.521,-27.760,35.953,-150.7835,-25.0572,0.0000
C01718=22.579,-30.435,37.285,-150.7779,-25.2528,0.0000
C01719=24.854,-33.391,38.288,-150.7317,-25.4864,0.0000
C01720=26.846,-36.198,38.776,-150.7234,-25.7631,0.0000
C01721=27.365,-39.186,39.032,-151.4360,-26.5279,0.0000
C01722=26.283,-41.963,39.238,-153.0110,-27.6459,0.0000
C01723=23.816,-43.952,39.446,-155.2383,-28.7415,0.0000
C01724=20.745,-45.492,39.582,-157.7360,-29.5707,0.0000
C01725=17.499,-46.837,39.582,-144.1323,6.6582,0.0000
C01726=14.238,-47.919,39.446,-143.0124,4.6080,0.0000
C01727=11.087,-48.257,39.238,-142.1966,2.5124,0.0000
C01728=8.359,-47.059,39.032,-141.8025,0.7627,0.0000
C01729=6.613,-44.579,38.776,-141.7735,-0.2340,0.0000
C01730=6.036,-41.186,38.288,-141.9501,-0.4472,0.0000
C01731=5.555,-37.486,37.285,-142.1271,-0.6052,0.0000
C01732=5.119,-34.140,35.953,-142.2518,-0.7560,0.0000
C01733=4.702,-31.601,34.645,-142.3126,-0.9188,0.0000
C01734=3.979,-30.109,33.696,-142.3127,-1.2565,0.0000
C01735=2.386,-29.720,33.319,-142.2773,-2.0340,0.0000
C01736=1.048,-29.759,33.303,-142.2483,-1.8474,0.0000
C01737=0.000,-29.775,33.314,-142.2164,-0.0017,0.0000
C01738=0.000,-29.775,33.314,-142.2164,-0.0017,0.0000
C01739=-1.048,-29.759,33.303,-142.2483,1.8478,0.0000
C01740=-2.386,-29.720,33.320,-142.2773,2.0334,0.0000
C01741=-3.979,-30.109,33.696,-142.3128,1.2560,0.0000
C01742=-4.702,-31.601,34.645,-142.3126,0.9184,0.0000
C01743=-5.119,-34.140,35.953,-142.2518,0.7556,0.0000
C01744=-5.555,-37.486,37.285,-142.1271,0.6048,0.0000
C01745=-6.036,-41.186,38.288,-141.9501,0.4468,0.0000
C01746=-6.613,-44.579,38.776,-141.7735,0.2335,0.0000
C01747=-8.359,-47.059,39.032,-141.8026,-0.7631,0.0000
C01748=-11.087,-48.257,39.238,-142.1966,-2.5126,0.0000
C01749=-14.238,-47.919,39.446,-143.0124,-4.6080,0.0000
C01750=-17.499,-46.837,39.582,-144.1323,-6.6582,0.0000
C01751=-20.745,-45.492,39.582,-157.7361,29.5707,0.0000
C01752=-23.816,-43.952,39.446,-155.2383,28.7414,0.0000
C01753=-26.283,-41.963,39.238,-153.0108,27.6458,0.0000
C01754=-27.365,-39.186,39.032,-151.4357,26.5277,0.0000
C01755=-26.846,-36.198,38.776,-150.7231,25.7628,0.0000
C01756=-24.854,-33.391,38.288,-150.7313,25.4860,0.0000
C01757=-22.579,-30.435,37.285,-150.7776,25.2525,0.0000
C01758=-20.521,-27.760,35.953,-150.7832,25.0569,0.0000
C01759=-19.020,-25.670,34.645,-150.7252,24.8912,0.0000
C01760=-18.476,-24.104,33.696,-150.4961,24.6252,0.0000
C01761=-19.328,-22.702,33.319,-149.9416,24.0332,0.0000
C01762=-20.302,-21.784,33.303,-150.0418,24.1985,0.0000
C01763=-21.054,-21.054,33.314,-151.2689,25.6714,0.0000
C01764=-21.784,-20.302,33.303,-152.5850,27.0967,0.0000
C01765=-22.702,-19.328,33.320,-152.7415,27.2229,0.0000
C01766=-24.104,-18.476,33.696,-152.2255,26.5953,0.0000
C01767=-25.670,-19.020,34.645,-151.9896,26.3319,0.0000
C01768=-27.760,-20.521,35.953,-151.8233,26.2426,0.0000
C01769=-30.435,-22.579,37.285,-151.6099,26.2022,0.0000
C01770=-33.391,-24.854,38.288,-151.3459,26.1884,0.0000
C01771=-36.198,-26.846,38.776,-151.0443,26.1304,0.0000
C01772=-39.186,-27.365,39.032,-150.3874,25.3280,0.0000
C01773=-41.963,-26.283,39.238,-149.5519,23.7038,0.0000
C01774=-43.952,-23.816,39.446,-148.8699,21.5457,0.0000
C01775=-45.492,-20.745,39.582,-148.4870,19.2399,0.0000
C01776=-46.837,-17.499,39.582,171.8030,35.5888,0.0000
C01777=-47.919,-14.238,39.446,174.2382,36.8483,0.0000
C01778=-48.257,-11.087,39.238,176.8215,37.7607,0.0000
C01779=-47.059,-8.359,39.032,179.0296,38.1935,0.0000
C01780=-44.579,-6.613,38.776,-179.7021,38.2262,0.0000
C01781=-41.186,-6.036,38.288,-179.4321,38.0486,0.0000
C01782=-37.486,-5.555,37.285,-179.2333,37.8704,0.0000
C01783=-34.140,-5.119,35.953,-179.0439,37.7444,0.0000
C01784=-31.601,-4.702,34.645,-178.8390,37.6817,0.0000
C01785=-30.109,-3.979,33.696,-178.4123,37.6766,0.0000
C01786=-29.720,-2.386,33.319,-177.4291,37.6947,0.0000
C01787=-29.759,-1.048,33.303,-177.6640,37.7286,0.0000
C01788=-29.775,0.000,33.314,-179.9979,37.7836,0.0000
C01789=-29.759,1.048,33.303,177.6635,37.7286,0.0000
C01790=-29.720,2.386,33.320,177.4299,37.6948,0.0000
C01791=-30.109,3.979,33.696,178.4130,37.6766,0.0000
C01792=-31.601,4.702,34.645,178.8395,37.6817,0.0000
C01793=-34.140,5.119,35.953,179.0444,37.7443,0.0000
C01794=-37.486,5.555,37.285,179.2338,37.8704,0.0000
C01795=-41.186,6.036,38.288,179.4326,38.0485,0.0000
C01796=-44.579,6.613,38.776,179.7027,38.2261,0.0000
C01797=-47.059,8.359,39.032,-179.0291,38.1934,0.0000
C01798=-48.257,11.087,39.238,-176.8212,37.7607,0.0000
C01799=-47.919,14.238,39.446,-174.2381,36.8483,0.0000
C01800=-46.837,17.499,39.582,-171.8030,35.5888,0.0000
C01801=-45.492,20.745,39.582,148.4871,19.2399,0.0000
C01802=-43.952,23.816,39.446,148.8700,21.5457,0.0000
C01803=-41.963,26.283,39.238,149.5520,23.7040,0.0000
C01804=-39.186,27.365,39.032,150.3876,25.3284,0.0000
C01805=-36.198,26.846,38.776,151.0446,26.1308,0.0000
C01806=-33.391,24.854,38.288,151.3462,26.1888,0.0000
C01807=-30.435,22.579,37.285,151.6102,26.2026,0.0000
C01808=-27.760,20.521,35.953,151.8236,26.2429,0.0000
C01809=-25.670,19.020,34.645,151.9899,26.3322,0.0000
C01810=-24.104,18.476,33.696,152.2258,26.5957,0.0000
C01811=-22.702,19.328,33.319,152.7420,27.2234,0.0000
C01812=-21.784,20.302,33.303,152.5848,27.0964,0.0000
C01813=-21.054,21.054,33.314,151.2712,25.6741,0.0000
C01814=-20.302,21.784,33.303,150.0415,24.1982,0.0000
C01815=-19.328,22.702,33.320,149.9420,24.0337,0.0000
C01816=-18.476,24.104,33.696,150.4965,24.6256,0.0000
C01817=-19.020,25.670,34.645,150.7255,24.8916,0.0000
C01818=-20.521,27.760,35.953,150.7835,25.0572,0.0000
C01819=-22.579,30.435,37.285,150.7779,25.2528,0.0000
C01820=-24.854,33.391,38.288,150.7317,25.4864,0.0000
C01821=-26.846,36.198,38.776,150.7234,25.7631,0.0000
C01822=-27.365,39.186,39.032,151.4360,26.5279,0.0000
C01823=-26.283,41.963,39.238,153.0110,27.6459,0.0000
C01824=-23.816,43.952,39.446,155.2383,28.7415,0.0000
C01825=-20.745,45.492,39.582,157.7360,29.5707,0.0000
C01826=-17.499,46.837,39.582,144.1323,-6.6582,0.0000
C01827=-14.238,47.919,39.446,143.0124,-4.6080,0.0000
C01828=-11.087,48.257,39.238,142.1966,-2.5126,0.0000
C01829=-8.359,47.059,39.032,141.8026,-0.7631,0.0000
C01830=-6.613,44.579,38.776,141.7735,0.2335,0.0000
C01831=-6.036,41.186,38.288,141.9501,0.4468,0.0000
C01832=-5.555,37.486,37.285,142.1271,0.6048,0.0000
C01833=-5.119,34.140,35.953,142.2518,0.7556,0.0000
C01834=-4.702,31.601,34.645,142.3126,0.9184,0.0000
C01835=-3.979,30.109,33.696,142.3128,1.2560,0.0000
C01836=-2.386,29.720,33.320,142.2773,2.0334,0.0000
C01837=-1.048,29.759,33.303,142.2483,1.8478,0.0000
C01838=0.000,29.775,33.314,142.2164,-0.0017,0.0000
C01839=0.000,28.557,35.146,142.5588,-0.0019,0.0000
C01840=0.937,28.545,35.134,142.5890,-1.7842,0.0000
C01841=2.198,28.517,35.152,142.6175,-2.0226,0.0000
C01842=3.753,28.963,35.561,142.6489,-1.2621,0.0000
C01843=4.437,30.601,36.587,142.6403,-0.9464,0.0000
C01844=4.837,33.354,37.988,142.5630,-0.7968,0.0000
C01845=5.276,36.942,39.399,142.4114,-0.6483,0.0000
C01846=5.763,40.861,40.447,142.1988,-0.4901,0.0000
C01847=6.331,44.425,40.953,141.9838,-0.2821,0.0000
C01848=8.101,47.028,41.216,141.9856,0.7519,0.0000
C01849=10.888,48.294,41.429,142.3842,2.5834,0.0000
C01850=14.116,47.960,41.642,143.2501,4.7750,0.0000
C01851=17.458,46.852,41.781,144.4494,6.9027,0.0000
C01852=20.785,45.474,41.781,158.1935,-29.5465,0.0000
C01853=23.932,43.894,41.642,155.5676,-28.7162,0.0000
C01854=26.450,41.848,41.429,153.2254,-27.5825,0.0000
C01855=27.526,38.982,41.216,151.5884,-26.4054,0.0000
C01856=26.937,35.890,40.953,150.8737,-25.5952,0.0000
C01857=24.818,32.968,40.447,150.9187,-25.2988,0.0000
C01858=22.391,29.853,39.399,150.9952,-25.0430,0.0000
C01859=20.165,27.005,37.988,151.0253,-24.8325,0.0000
C01860=18.500,24.775,36.587,150.9902,-24.6672,0.0000
C01861=17.826,23.134,35.561,150.7832,-24.4137,0.0000
C01862=18.610,21.719,35.152,150.2430,-23.8337,0.0000
C01863=19.522,20.847,35.134,150.3788,-24.0393,0.0000
C01864=20.193,20.193,35.146,151.5662,-25.4586,0.0000
C01865=20.846,19.522,35.134,152.8377,-26.8337,0.0000
C01866=21.719,18.610,35.152,153.0301,-26.9999,0.0000
